# B&R Automation Studio project NAELD004C00R10L518F00 (part 41)

#### InputRef.var - Do Not Change!!!
```iecst
(*2021-08-01*)
(**)
(*General*)
VAR
	p_eAct : REFERENCE TO eHermesAction;
	p_udiRstErr : REFERENCE TO UDINT;
	p_bPrep : REFERENCE TO BOOL;
	p_bEn : REFERENCE TO BOOL;
	p_bDis : REFERENCE TO BOOL;
END_VAR
(**)
(*Configuration*)
VAR
	p_tyParam : REFERENCE TO tyHermesDSParam;
	p_sIPAddr : REFERENCE TO STRING[15];
	pa_usiMacAddr : REFERENCE TO ARRAY[0..5] OF USINT;
	p_tyDTStructure : REFERENCE TO DTStructure;
	p_dtCurrDT : REFERENCE TO DATE_AND_TIME;
	p_sMcId : REFERENCE TO STRING[80];
END_VAR
(**)
(*Input*)
VAR
	p_bRdySnd : REFERENCE TO BOOL;
	p_bSndCompl : REFERENCE TO BOOL;
	p_bSndIncompl : REFERENCE TO BOOL;
	p_bSndNotStart : REFERENCE TO BOOL;
	p_bBAWidthEn : REFERENCE TO BOOL; (*Board Available Check Width*)
	p_bBASltEn : REFERENCE TO BOOL; (*Board Available Check Slot*)
	p_bBFWidthEn : REFERENCE TO BOOL; (*Board Forecast Check Width*)
	p_bBFSltEn : REFERENCE TO BOOL; (*Board Forecast Check Slot*)
	p_sRecipeNm : REFERENCE TO STRING[254];
	p_sForecastId : REFERENCE TO STRING[80];
	p_sBoardId : REFERENCE TO STRING[36];
	p_sInterfaceId : REFERENCE TO STRING[80];
	p_sVersion : REFERENCE TO STRING[7];
	p_eFailedBoard : REFERENCE TO eHermesFailedBoard;
	p_eFlippedBoard : REFERENCE TO eHermesFlippedBoard;
	p_sTopBarcode : REFERENCE TO STRING[254];
	p_sBottomBarcode : REFERENCE TO STRING[254];
	p_rLength : REFERENCE TO REAL;
	p_rThickness : REFERENCE TO REAL;
	p_rConveyorSpeed : REFERENCE TO REAL;
	p_rTopClearanceHeight : REFERENCE TO REAL;
	p_rBottomClearanceHeight : REFERENCE TO REAL;
	p_rWeight : REFERENCE TO REAL;
	p_sWorkOrderId : REFERENCE TO STRING[80];
	p_sBatchId : REFERENCE TO STRING[80];
	p_diWidthInUM : REFERENCE TO DINT;
	p_diMinSltValue : REFERENCE TO DINT;
	p_diMaxSltValue : REFERENCE TO DINT;
	p_diPitch : REFERENCE TO DINT;
	p_diTtlSlt : REFERENCE TO DINT;
	p_diSltToSltInUM : REFERENCE TO DINT;
	p_udiSndBffrSize : REFERENCE TO UDINT;
	p_udiRcvBffrSize : REFERENCE TO UDINT;
	p_udiAliveIdleTimeInSec : REFERENCE TO UDINT;
	p_tConnTimeOut : REFERENCE TO TIME;
	p_diTransferInTO : REFERENCE TO DINT;
	pa_tyXMLTableDataBrdAvl : REFERENCE TO ARRAY[0..200] OF tyXMLTableDat;
	p_iXMLTableDataBrdAvlTtlIdx : REFERENCE TO INT;
	p_bNewBrdAvlFirstZone : REFERENCE TO BOOL;
	p_bNewBrdAvlLastZone : REFERENCE TO BOOL;
	p_bOpsRun : REFERENCE TO BOOL;
	p_bInterruptSen : REFERENCE TO BOOL;
	p_udiFileKeepDay : REFERENCE TO UDINT;
	p_udiRetainDataAddr : REFERENCE TO UDINT;
	p_udiRetainDataLen : REFERENCE TO UDINT;
	p_sRetainFileName : REFERENCE TO STRING[80];
	p_sProgNm : REFERENCE TO STRING[15];
	p_bNtSettingsLoadDone : REFERENCE TO BOOL;
	p_bRmtPrep : REFERENCE TO BOOL;
	p_bRmtEn : REFERENCE TO BOOL;
	p_bSvyPrep : REFERENCE TO BOOL;
	p_bSvyEn : REFERENCE TO BOOL;
	p_bOpsGConv1HvBrd : REFERENCE TO BOOL;
	p_bAllZonesEmpty : REFERENCE TO BOOL;
	p_bFirstZoneHaveBoard : REFERENCE TO BOOL;
	p_tyUSBoardArrivedData : REFERENCE TO tyHermesBoardAvailable;
	p_rMcCycleTm : REFERENCE TO REAL;
	p_rAWCycleTm : REFERENCE TO REAL;
	p_bInitDone : REFERENCE TO BOOL;
	p_tyHermesConfiguration : REFERENCE TO tyHermesConfiguration;
	p_bUSHermesStopTransport : REFERENCE TO BOOL;
	p_bRcvBoardInfo : REFERENCE TO BOOL;
	p_tyBoardInfoData : REFERENCE TO tyHermesSendBoardInfo;
	p_tySendWorkOrderData : REFERENCE TO tyHermesSendWorkOrderInfo;
	p_bUSHermesTransporting : REFERENCE TO BOOL;
	p_bReplyWorkOrderInfo : REFERENCE TO BOOL;
	p_bSendBoardForecast : REFERENCE TO BOOL;
	p_bClearWorkOrder : REFERENCE TO BOOL;
	p_bFirstZoneEndSen : REFERENCE TO BOOL;
	p_bNewProduct : REFERENCE TO BOOL;
	p_bNewWidth : REFERENCE TO BOOL;
	p_bInternalUse : REFERENCE TO BOOL;
	p_sInternalRcv : REFERENCE TO STRING[65535];
	p_tyDI : REFERENCE TO tyDigitalInput;
	p_usiProdRcpCurrRcp1McMod : REFERENCE TO USINT;
	p_usiSelProdRcpStep : REFERENCE TO USINT;
END_VAR
(**)
(*Dummy*)
VAR
	p_sFoundAddressTop : REFERENCE TO STRING[254];
	p_sFoundAddressBottom : REFERENCE TO STRING[254];
END_VAR
```

#### Local.var - Do Not Change!!!
```iecst
(*2021-08-01*)
(**)
(*Local Action, State & Status*)
VAR
	eAct : eHermesAction := HermesActIdle;
	eStat : eHermesAction := HermesActIdle;
	eMainStatus : eFBStatus := Idle;
	eStatus : eFBStatus := Idle;
	eStatus1 : eFBStatus := Idle;
	eStatus2 : eFBStatus := Idle;
	eStatus3 : eFBStatus := Idle;
	udiStatus : UDINT := 0;
	udiStatus1 : UDINT := 0;
	udiStatus2 : UDINT := 0;
	udiStatus3 : UDINT := 0;
	udiStatus4 : UDINT := 0;
	sStatTxt : STRING[200] := '';
	a_sStatText : ARRAY[0..50] OF STRING[200] := ['Idling','Background Starting Operations','Background Stopping Operations','Deleting Old Log File','Creating Directory','Writing Retain File','Reading Retain File','Saving Configuration',43('')];
END_VAR
(**)
(*Local Alarm*)
VAR
	tyAlmData : tyAlmDat;
	tyAlmData1 : tyAlmDat;
	tyAlmData2 : tyAlmDat;
	tyAlmData3 : tyAlmDat;
	tyAlmData4 : tyAlmDat;
	a_tyAlmText : ARRAY[10000..10199] OF tyAlmTxt := [(sAlmText:='Invalid Ident While Creating Server',sRcyText:='Problem Occurred In The TCP/IP Connection. Check The Connection And Try To Reconnect.'),(sAlmText:='Setting Keep Alive Interval Time Error While Creating Server',sRcyText:='Unable To Establish Connection Between Machine. Check For Setting And Resume Operation.'),(sAlmText:='Setting Keep Alive Idle Time Error While Creating Server',sRcyText:='Unable To Establish Connection Between Machine. Check For Setting And Resume Operation.'),(sAlmText:='Setting Keep Alive Count Error While Creating Server',sRcyText:='Unable To Establish Connection Between Machine. Check For Setting And Resume Operation.'),(sAlmText:='Setting Keep Alive Error While Creating Server',sRcyText:='Unable To Establish Connection Between Machine. Check For Setting And Resume Operation.'),(sAlmText:='Setting Receive Buffer Error While Creating Server',sRcyText:='Unable To Establish Connection Between Machine. Check For Setting And Resume Operation.'),(sAlmText:='Setting Send Buffer Error While Creating Server',sRcyText:='Unable To Establish Connection Between Machine. Check For Setting And Resume Operation.'),(sAlmText:='Setting No Waiting Error While Creating Server',sRcyText:='Unable To Establish Connection Between Machine. Check For Setting And Resume Operation.'),(sAlmText:='TCP Open Port Error While Creating Server',sRcyText:='Problem Occurred In The TCP/IP Connection. Check The Connection And Try To Reconnect.'),(sAlmText:='Closing TCP Error While Creating Server',sRcyText:='Problem Occurred In The TCP/IP Connection. Check The Connection And Try To Reconnect.'),(sAlmText:='Invalid Ident While Listening Client',sRcyText:='There Was A Problem Connecting To The Server. The Server May Not Exist or It is Unavailable At This Time. Check The Connection and Try Again.'),0,(sAlmText:='DS Hermes Connection Lost',sRcyText:='There Was A Problem Connecting To The Server. The Server May Not Exist or It is Unavailable At This Time. Check The Connection and Try Again.'),0,(sAlmText:='Invalid Ident While Receiving Data',sRcyText:='Problem Occurred In The TCP/IP Connection. Check The Connection And Try To Reconnect.'),(sAlmText:='TCP Receive Data Error While Receiving Data',sRcyText:='Problem Occurred In The TCP/IP Connection. Check The Connection And Try To Reconnect.'),(sAlmText:='Receive BoardAvailable While Downstream In Not Connected State',sRcyText:='Receive Illegal Message.'),(sAlmText:='Receive RevokeBoardAvailable While Downstream In Not Connected State',sRcyText:='Receive Illegal Message.'),(sAlmText:='Receive MachineReady While Downstream In Not Connected State',sRcyText:='Receive Illegal Message.'),(sAlmText:='Receive RevokeMachineReady While Downstream In Not Connected State',sRcyText:='Receive Illegal Message.'),(sAlmText:='Receive StartTransport While Downstream In Not Connected State',sRcyText:='Receive Illegal Message.'),(sAlmText:='Receive StopTransport While Downstream In Not Connected State',sRcyText:='Receive Illegal Message.'),(sAlmText:='Receive TransportFinished While Downstream In Not Connected State',sRcyText:='Receive Illegal Message.'),(sAlmText:='Receive BoardForecast While Downstream In Not Connected State',sRcyText:='Receive Illegal Message.'),(sAlmText:='Receive ServiceDescription While Downstream In Service Description State',sRcyText:='Receive Illegal Message.'),(sAlmText:='Receive BoardAvailable While Downstream In Service Description State',sRcyText:='Receive Illegal Message.'),(sAlmText:='Receive RevokeBoardAvailable While Downstream In Service Description State',sRcyText:='Receive Illegal Message.'),(sAlmText:='Receive MachineReady While Downstream In Service Description State',sRcyText:='Receive Illegal Message.'),(sAlmText:='Receive RevokeMachineReady While Downstream In Service Description State',sRcyText:='Receive Illegal Message.'),(sAlmText:='Receive StartTransport While Downstream In Service Description State',sRcyText:='Receive Illegal Message.'),(sAlmText:='Receive StopTransport While Downstream In Service Description State',sRcyText:='Receive Illegal Message.'),(sAlmText:='Receive TransportFinished While Downstream In Service Description State',sRcyText:='Receive Illegal Message.'),(sAlmText:='Receive BoardForecast While Downstream In Service Description State',sRcyText:='Receive Illegal Message.'),(sAlmText:='Receive ServiceDescription While Downstream In Not Available Not Ready State',sRcyText:='Receive Illegal Message.'),(sAlmText:='Receive BoardAvailable While Downstream In Not Available Not Ready State',sRcyText:='Receive Illegal Message.'),(sAlmText:='Receive RevokeBoardAvailable While Downstream In Not Available Not Ready State',sRcyText:='Receive Illegal Message.'),(sAlmText:='Receive RevokeMachineReady While Downstream In Not Available Not Ready State',sRcyText:='Receive Illegal Message.'),(sAlmText:='Receive StartTransport While Downstream In Not Available Not Ready State',sRcyText:='Receive Illegal Message.'),(sAlmText:='Receive StopTransport While Downstream In Not Available Not Ready State',sRcyText:='Receive Illegal Message.'),(sAlmText:='Receive TransportFinished While Downstream In Not Available Not Ready State',sRcyText:='Receive Illegal Message.'),(sAlmText:='Receive BoardForecast While Downstream In Not Available Not Ready State',sRcyText:='Receive Illegal Message.'),(sAlmText:='Receive ServiceDescription While Downstream In Board Available State',sRcyText:='Receive Illegal Message.'),(sAlmText:='Receive BoardAvailable While Downstream In Board Available State',sRcyText:='Receive Illegal Message.'),(sAlmText:='Receive RevokeBoardAvailable While Downstream In Board Available State',sRcyText:='Receive Illegal Message.'),(sAlmText:='Receive RevokeMachineReady While Downstream In Board Available State',sRcyText:='Receive Illegal Message.'),(sAlmText:='Receive StartTransport While Downstream In Board Available State',sRcyText:='Receive Illegal Message.'),(sAlmText:='Receive StopTransport While Downstream In Board Available State',sRcyText:='Receive Illegal Message.'),(sAlmText:='Receive TransportFinished While Downstream In Board Available State',sRcyText:='Receive Illegal Message.'),(sAlmText:='Receive BoardForecast While Downstream In Board Available State',sRcyText:='Receive Illegal Message.'),(sAlmText:='Receive ServiceDescription While Downstream In Machine Ready State',sRcyText:='Receive Illegal Message.'),(sAlmText:='Receive BoardAvailable While Downstream In Machine Ready State',sRcyText:='Receive Illegal Message.'),(sAlmText:='Receive RevokeBoardAvailable While Downstream In Machine Ready State',sRcyText:='Receive Illegal Message.'),(sAlmText:='Receive MachineReady While Downstream In Machine Ready State',sRcyText:='Receive Illegal Message.'),(sAlmText:='Receive StopTransport While Downstream In Machine Ready State',sRcyText:='Receive Illegal Message.'),(sAlmText:='Receive TransportFinished While Downstream In Machine Ready State',sRcyText:='Receive Illegal Message.'),(sAlmText:='Receive BoardForecast While Downstream In Machine Ready State',sRcyText:='Receive Illegal Message.'),(sAlmText:='Receive ServiceDescription While Downstream In Available And Ready State',sRcyText:='Receive Illegal Message.'),(sAlmText:='Receive BoardAvailable While Downstream In Available And Ready State',sRcyText:='Receive Illegal Message.'),(sAlmText:='Receive RevokeBoardAvailable While Downstream In Available And Ready State',sRcyText:='Receive Illegal Message.'),(sAlmText:='Receive MachineReady While Downstream In Available And Ready State',sRcyText:='Receive Illegal Message.'),(sAlmText:='Receive StopTransport While Downstream In Available And Ready State',sRcyText:='Receive Illegal Message.'),(sAlmText:='Receive TransportFinished While Downstream In Available And Ready State',sRcyText:='Receive Illegal Message.'),(sAlmText:='Receive BoardForecast While Downstream In Available And Ready State',sRcyText:='Receive Illegal Message.'),(sAlmText:='Receive ServiceDescription While Downstream In Transporting State',sRcyText:='Receive Illegal Message.'),(sAlmText:='Receive BoardAvailable While Downstream In Transporting State',sRcyText:='Receive Illegal Message.'),(sAlmText:='Receive RevokeBoardAvailable While Downstream In Transporting State',sRcyText:='Receive Illegal Message.'),(sAlmText:='Receive MachineReady While Downstream In Transporting State',sRcyText:='Receive Illegal Message.'),(sAlmText:='Receive RevokeMachineReady While Downstream In Transporting State',sRcyText:='Receive Illegal Message.'),(sAlmText:='Receive StartTransport While Downstream In Transporting State',sRcyText:='Receive Illegal Message.'),(sAlmText:='Receive TransportFinished While Downstream In Transporting State',sRcyText:='Receive Illegal Message.'),(sAlmText:='Receive BoardForecast While Downstream In Transporting State',sRcyText:='Receive Illegal Message.'),(sAlmText:='Receive ServiceDescription While In Transport Finished State',sRcyText:='Receive Illegal Message.'),(sAlmText:='Receive BoardAvailable While In Transport Finished State',sRcyText:='Receive Illegal Message.'),(sAlmText:='Receive RevokeBoardAvailable While In Transport Finished State',sRcyText:='Receive Illegal Message.'),(sAlmText:='Receive MachineReady While In Transport Finished State',sRcyText:='Receive Illegal Message.'),(sAlmText:='Receive RevokeMachineReady While In Transport Finished State',sRcyText:='Receive Illegal Message.'),(sAlmText:='Receive StartTransport While In Transport Finished State',sRcyText:='Receive Illegal Message.'),(sAlmText:='Receive TransportFinished While In Transport Finished State',sRcyText:='Receive Illegal Message.'),(sAlmText:='Receive BoardForecast While In Transport Finished State',sRcyText:='Receive Illegal Message.'),(sAlmText:='Receive ServiceDescription While Downstream In Transport Stopped State',sRcyText:='Receive Illegal Message.'),(sAlmText:='Receive BoardAvailable While Downstream In Transport Stopped State',sRcyText:='Receive Illegal Message.'),(sAlmText:='Receive RevokeBoardAvailable While Downstream In Transport Stopped State',sRcyText:='Receive Illegal Message.'),(sAlmText:='Receive MachineReady While Downstream In Transport Stopped State',sRcyText:='Receive Illegal Message.'),(sAlmText:='Receive RevokeMachineReady While Downstream In Transport Stopped State',sRcyText:='Receive Illegal Message.'),(sAlmText:='Receive StartTransport While Downstream In Transport Stopped State',sRcyText:='Receive Illegal Message.'),(sAlmText:='Receive StopTransport While Downstream In Transport Stopped State',sRcyText:='Receive Illegal Message.'),(sAlmText:='LaneId Mismatch While Checking Service Description',sRcyText:='The LaneId Value Does Not Match. Change The Value And Resend The Value.'),(sAlmText:='MachineId Missing While Checking Service Description',sRcyText:='Missing Input Value For MachineId. Fill Up The Value And Resend.'),(sAlmText:='LandId Out Of Range While Checking Service Description',sRcyText:='LaneId Does Not Fall Within The Expected Range.'),(sAlmText:='LandId Missing While Checking Service Description',sRcyText:='Missing Input Value For LaneId. Fill Up The Value And Resend.'),(sAlmText:='Version Missing While Checking Service Description',sRcyText:='Missing Input Value For Version. Fill Up The Value And Resend.'),(sAlmText:='SupportedFeatures Missing While Checking Service Description',sRcyText:='Missing Input Value For SupportedFeatures. Fill Up The Value And Resend.'),(sAlmText:='NotificationCode Out Of Range While Checking Notification',sRcyText:='NotificationCode Does Not Fall Within The Expected Range.'),(sAlmText:='NotificationCode Missing While Checking Notification',sRcyText:='Missing Input Value For NotificationCode. Fill Up The Value And Resend.'),(sAlmText:='Severity Missing While Checking Notification',sRcyText:='Missing Input Value For Severity. Fill Up The Value And Resend.'),(sAlmText:='Description Missing While Checking Notification',sRcyText:='Missing Input Value For Description. Fill Up The Value And Resend.'),2((0)),(sAlmText:='FailedBoard Missing While Checking Machine Ready',sRcyText:='Missing Input Value For FailedBoard. Fill Up The Value And Resend.'),(sAlmText:='TransferState Missing While Checking Stop Transport',sRcyText:='Missing Input Value For TransferState. Fill Up The Value And Resend.'),(sAlmText:='BoardId Missing While Checking Stop Transport',sRcyText:='Missing Input Value For BoardId. Fill Up The Value And Resend.'),(sAlmText:='BoardId Missing While Checking Start Transport',sRcyText:='Missing Input Value For BoardId. Fill Up The Value And Resend.'),(sAlmText:='Barcode Missing While Checking Query Board Info',sRcyText:='Missing Input Value For BoardId. Fill Up The Value And Resend.'),(0),(sAlmText:='BoardId Mismatch While Checking Start Transport & Stop Transport',sRcyText:='The BoardId Value Does Not Match. Change The Value And Resend The Value.'),(sAlmText:='BoardId Missing While Checking Start Transport & Stop Transport',sRcyText:='Missing Input Value For BoardId. Fill Up The Value And Resend.'),(sAlmText:='Service Description Interchange Time Out',sRcyText:='Timeout Expired Before Operation Completed. Reset And Resume Operation.'),(sAlmText:='Transport Time Out',sRcyText:='Timeout Expired Before Operation Completed. Reset And Resume Operation.'),(sAlmText:='Receive TransportFinished While Downstream In Transport Stopped State',sRcyText:='Receive Illegal Message.'),(sAlmText:='Receive BoardForecast While Downstream In Transport Stopped State',sRcyText:='Receive Illegal Message.'),(sAlmText:='Stop Transport Request To Send From Downstream Hermes',sRcyText:='Sending Illegal Message.'),(sAlmText:='Get Directory Info Error While Deleting Old Log',sRcyText:='An Error Was Encountered While Getting Directory Info. Please Contact Nutek For A Possible Solution.'),(sAlmText:='Directory Read Error While Deleting Old Log',sRcyText:='An Error Was Encountered While Reading Directory. Please Contact Nutek For A Possible Solution.'),(sAlmText:='File Delete Error While Deleting Old Log',sRcyText:='An Error Was Encountered While Trying To Delete File. Please Contact Nutek For A Possible Solution.'),(sAlmText:='File Open Error While Reading Retain File',sRcyText:='An Error Was Encountered While Trying To Open File. Please Contact Nutek For A Possible Solution.'),(sAlmText:='File Read Error While Reading Retain File',sRcyText:='An Error Was Encountered While Trying To Read File. Please Contact Nutek For A Possible Solution.'),(sAlmText:='File Close Error While Reading Retain File',sRcyText:='An Error Was Encountered While Trying To Close File. Please Contact Nutek For A Possible Solution.'),(sAlmText:='File Open Error While Writing Retain File',sRcyText:='An Error Was Encountered While Trying To Open File. Please Contact Nutek For A Possible Solution.'),(sAlmText:='File Create Error While Writing Retain File',sRcyText:='An Error Was Encountered While Trying To Create File. Please Contact Nutek For A Possible Solution.'),(sAlmText:='File Write Error While Writing Retain File',sRcyText:='An Error Was Encountered While Trying To Write File. Please Contact Nutek For A Possible Solution.'),(sAlmText:='File Close Error While Writing Retain File',sRcyText:='An Error Was Encountered While Trying To Close File. Please Contact Nutek For A Possible Solution.'),(sAlmText:='Directory Does Not Exist While Writing Retain File',sRcyText:='The Directory Does Not Exist. Please Contact Nutek For A Possible Solution.'),10((0)),(sAlmText:='Check Alive Time Out',sRcyText:='Timeout Expired Before Operation Completed. Reset And Resume Operation.'),(sAlmText:='Waiting Check Alive Time Out',sRcyText:='Timeout Expired Before Operation Completed. Reset And Resume Operation.'),(sAlmText:='Check Alive Id Mismatch',sRcyText:='The Check Alive Id Value Does Not Match. Change The Value And Resend The Value.'),(sAlmText:='Machine Ready Request To Send From Downstream Hermes',sRcyText:='Sending Illegal Message.'),(sAlmText:='Revoke Machine Ready Request To Send From Downstream Hermes',sRcyText:='Sending Illegal Message.'),(sAlmText:='Start Transport Request To Send From Downstream Hermes',sRcyText:='Sending Illegal Message.'),(sAlmText:='Set Configuration Request To Send From Downstream Hermes',sRcyText:='Sending Illegal Message.'),(sAlmText:='Get Configuration Request To Send From Downstream Hermes',sRcyText:='Sending Illegal Message.'),(sAlmText:='Current Configuration Request To Send From Downstream Hermes',sRcyText:='Sending Illegal Message.'),(sAlmText:='Board Forecast Request To Send From Downstream Hermes',sRcyText:='Sending Illegal Message.'),(sAlmText:='Query Board Info Request To Send From Downstream Hermes',sRcyText:='Sending Illegal Message.'),(sAlmText:='Invalid Ident While Sending Data',sRcyText:='Invalid Ident Value.'),(sAlmText:='TCP Retry Send Data Error While Sending Data',sRcyText:='Problem Occurred In The TCP/IP Connection. Check The Connection And Try To Reconnect.'),(sAlmText:='TCP Send Data Error',sRcyText:='Problem Occurred In The TCP/IP Connection. Check The Connection And Try To Reconnect.'),(sAlmText:='Invalid Ident While Closing TCP',sRcyText:='Invalid Ident Value.'),(sAlmText:='Closing TCP Error',sRcyText:='Problem Occurred In The TCP/IP Connection. Check The Connection And Try To Reconnect.'),(sAlmText:='File Open Error While Writing Log',sRcyText:='An Error Was Encountered While Trying To Open File. Please Contact Nutek For A Possible Solution.'),(sAlmText:='File Create Error While Writing Log',sRcyText:='An Error Was Encountered While Trying To Create File. Please Contact Nutek For A Possible Solution.'),(sAlmText:='Get File Info Error While Writing Log',sRcyText:='An Error Was Encountered While Getting File Info. Please Contact Nutek For A Possible Solution.'),(sAlmText:='File Write Error While Writing Log',sRcyText:='An Error Was Encountered While Trying To Write File. Please Contact Nutek For A Possible Solution.'),(sAlmText:='File Close Error While Writing Log',sRcyText:='An Error Was Encountered While Trying To Close File. Please Contact Nutek For A Possible Solution.'),(sAlmText:='Directory Does Not Exist While Writing Log',sRcyText:='The Directory Does Not Exist.Please Contact Nutek For A Possible Solution.'),(sAlmText:='Invalid Ident While Closing TCP',sRcyText:='Invalid Ident Value.'),(sAlmText:='Closing TCP Error',sRcyText:='Problem Occurred In The TCP/IP Connection. Check The Connection And Try To Reconnect.'),0,(sAlmText:='Board Jam At Sensor After Transfer Interrupted',sRcyText:='Pull Back Board From Downstream Machine'),0,(sAlmText:='Send Board Info Request To Send From Downstream Hermes',sRcyText:='Sending Illegal Message.'),(sAlmText:='Query Work Order Info Request To Send From Downstream Hermes',sRcyText:='Sending Illegal Message.'),(sAlmText:='Send Work Order Info Request To Send From Downstream Hermes',sRcyText:='Sending Illegal Message.'),(sAlmText:='Board Arrived Request To Send From Downstream Hermes',sRcyText:='Sending Illegal Message.'),(sAlmText:='Board departed Request To Send From Downstream Hermes',sRcyText:='Sending Illegal Message.'),(sAlmText:='Forecast Id Mismatch While Checking BoardForecast & Machine Ready',sRcyText:='The ForecastId Value Does Not Match. Change The Value And Resend The Value.'),(sAlmText:='Product Type Id Mismatch While Checking BoardForecast & Machine Ready',sRcyText:='The ProductTypetId Value Does Not Match. Change The Value And Resend The Value.'),(sAlmText:='Width Mismatch While Checking BoardForecast & Machine Ready',sRcyText:='The Width Value Does Not Match. Change The Value And Resend The Value.'),(sAlmText:='Query Top Barcode and Bottom Barcode found from different Recipes',sRcyText:='Please Check or Scan Again the PCB Barcode'),32(0)];
END_VAR
(**)
(*Local Output*)
VAR
	bConnected : BOOL;
	bHandshakeDone : BOOL;
	bSendOk : BOOL;
	bSearchTop : BOOL;
	bSearchBottom : BOOL;
	bFoundIndex : BOOL;
	bFoundTop : BOOL;
	bFoundBottom : BOOL;
	bFoundNothing : BOOL;
	bNewChangeOver : BOOL;
	bSendBFId : BOOL;
	bRstSendBFId : BOOL;
	bUSRdy : BOOL;
	bDSRdy : BOOL;
	bUSGdRdy : BOOL;
	bDSGdRdy : BOOL;
	bTransporting : BOOL;
	bStopTransport : BOOL;
	sInternalSnd : STRING[65535];
	bTransportFinishedSnd : BOOL;
	tyBoardDepartedInfo : tyHermesBoardAvailable;
END_VAR
(**)
(*Local Input*)
VAR
	udiRstErr : UDINT := 0;
	bPrep : BOOL := TRUE;
	bEn : BOOL := TRUE;
	bDis : BOOL := FALSE;
	tyParam : tyHermesDSParam;
	sIPAddr : STRING[15] := '192.168.0.100';
	a_usiMacAddr : ARRAY[0..5] OF USINT := [6(0)];
	tyDTStructure : DTStructure := (year:=2020,month:=11,day:=11,wday:=05,hour:=21,minute:=28,second:=30,millisec:=123,microsec:=456);
	dtCurrDT : DATE_AND_TIME := DT#2019-02-23-12:30:50;
	bRdySnd : BOOL := FALSE;
	bSndCompl : BOOL := FALSE;
	bSndInCompl : BOOL := FALSE;
	bSndNotStart : BOOL := FALSE;
	bFirstZoneEndSen : BOOL;
	bBAWidthEn : BOOL := TRUE; (*Board Available Check Width*)
	bBASltEn : BOOL := TRUE; (*Board Available Check Slot*)
	bBFWidthEn : BOOL := TRUE; (*Board Forecast Check Width*)
	bBFSltEn : BOOL := FALSE; (*Board Forecst Check Slot*)
	sForecastId : {REDUND_UNREPLICABLE} STRING[80] := '';
	sBoardId : STRING[36] := '';
	sMcId : STRING[80] := '';
	sInterfaceId : STRING[80] := '';
	sVersion : STRING[7] := '1.3';
	eFailedBoard : eHermesFailedBoard := HermesUnknownBoard;
	sRecipeNm : STRING[254] := '';
	eFlippedBoard : eHermesFlippedBoard := HermesFlippedBoardUnknownSide;
	sTopBarcode : STRING[254] := '';
	sBottomBarcode : STRING[254] := '';
	rLength : REAL := 0;
	rThickness : REAL := 0;
	rConveyorSpeed : REAL := 0;
	rTopClearanceHeight : REAL := 0;
	rBottomClearanceHeight : REAL := 0;
	rWeight : REAL := 0;
	sWorkOrderId : STRING[80] := '';
	sBatchId : STRING[80] := '';
	diWidthInUM : DINT := 0;
	diMinSltValue : DINT := 0;
	diMaxSltValue : DINT := 0;
	diPitch : DINT := 0;
	diTtlSlt : DINT := 0;
	diSltToSltInUM : DINT := 0;
	udiSndBffrSize : UDINT := 65536;
	udiRcvBffrSize : UDINT := 65536;
	udiAliveIdleTimeInSec : UDINT := 5;
	tConnTimeOut : TIME := T#30s;
	diTransferInTO : DINT := 30000;
	a_tyXMLTableDataBrdAvl : ARRAY[0..200] OF tyXMLTableDat;
	iXMLTableDataBrdAvlTtlIdx : INT := 0;
	bNewBrdAvl1 : BOOL := FALSE;
	bNewBrdAvl2 : BOOL := FALSE;
	bOpsRun : BOOL := FALSE;
	bInterruptSen : BOOL := FALSE;
	udiFileKeepDay : UDINT := 30;
	sRetainFileName : STRING[80] := 'BoardData.dat';
	sProgNm : STRING[15] := 'DSHermes';
	bNtSettingsLoadDone : BOOL := TRUE;
	bRmtPrep : BOOL := FALSE;
	bRmtEn : BOOL := FALSE;
	bSvyPrep : BOOL := FALSE;
	bSvyEn : BOOL := FALSE;
	bAllZonesEmpty : BOOL := FALSE;
	bFirstZoneHaveBoard : BOOL := FALSE;
	bInternalUse : BOOL;
	sInternalRcv : STRING[65535];
	rMachineCycleTime : REAL := 6000;
	rAutoWidthCycleTime : REAL := 30000;
	tyHermesCurrConfiguration : tyHermesConfiguration;
	tyBoardInfoData : tyHermesSendBoardInfo;
	tyUSBoardArrivedData : tyHermesBoardAvailable;
	bUSHermesStopTransport : BOOL;
	bRcvBoardInfo : BOOL;
	bUSHermesTransporting : BOOL;
	bOpsGConv1HvBrd : BOOL;
END_VAR
(**)
(*Local*)
VAR
	bRstErr : BOOL;
	udiRstErrOld : UDINT;
	bInitDone : BOOL;
	bInitialDone : BOOL;
	bRun : BOOL;
	bStop : BOOL;
	bRstConnection : BOOL;
	bRstState : BOOL;
	udiSvrIdent : UDINT;
	udiClntIdent : UDINT;
	udiClntIdentExtra : UDINT;
	udiXMLTableWriteIdx : UDINT;
	udiMsgSendBffr : UDINT;
	udiSndMsgLen : UDINT;
	sSnd : STRING[65535];
	sRcv : STRING[65535];
	a_tyXMLTableDataRcv : ARRAY[0..200] OF tyXMLTableDat;
	a_tyXMLTableDataSnd : ARRAY[0..200] OF tyXMLTableDat;
	a_eMsgSend : ARRAY[0..50] OF eHermesMsgType;
	tyMsgTypeRcv : tyHermesMsgType;
	tyCheckAliveSnd : tyHermesCheckAlive;
	tyCheckAlivePingSnd : tyHermesCheckAlive;
	tyCheckAlivePongSnd : tyHermesCheckAlive;
	tyCheckAliveRcv : tyHermesCheckAlive;
	tyCheckAlivePingRcv : tyHermesCheckAlive;
	tyCheckAlivePongRcv : tyHermesCheckAlive;
	tyServiceDescriptionSnd : tyHermesServiceDescription;
	tyServiceDescriptionRcv : tyHermesServiceDescription;
	tyNotificationSnd : tyHermesNotification;
	tyNotificationRcv : tyHermesNotification;
	tyBoardAvailableRcv : tyHermesBoardAvailable;
	tyBoardAvailableSnd : tyHermesBoardAvailable;
	a_tyBoardDepartedInfo : ARRAY[0..49] OF tyHermesBoardAvailable;
	tyMachineReady : tyHermesMachineReady;
	tyStartTransport : tyHermesStartTransport;
	tyStopTransport : tyHermesStopTransport;
	tyTransportFinished : tyHermesTransportFinished;
	tySetConfiguration : tyHermesSetConfiguration;
	tyCurrentConfiguration : tyHermesCurrentConfiguration;
	tyBoardForecastRcv : tyHermesBoardForecast;
	tyBoardForecastSnd : tyHermesBoardForecast;
	tyQueryBoardInfo : tyHermesQueryBoardInfo;
	tySendBoardInfo : tyHermesSendBoardInfo;
	fbCreateSvr : fbTCPCreateSvr;
	fbListen : fbTCPListen;
	fbRcv : fbTCPRcv;
	fbSend : fbTCPSnd;
	fbCloseSvr : fbTCPClose;
	fbCloseClnt : fbTCPClose;
	fbParseXMLTable : fbHermesParseXMLTable;
	fbParseBrdAvlExternal : fbHermesParseXMLTable;
	fbCheckAlive : fbHermesCheckAlive;
	fbCheckAliveSendPing : fbHermesCheckAliveSendPing;
	fbCheckAliveRcvPing : fbHermesCheckAliveRcvPing;
	fbSequenceDS : fbHermesSequenceDS;
	fbSequenceTO : fbHermesSequenceTO;
	eStatOld : eHermesAction := HermesActIdle;
	tyParamOld : tyHermesDSParam;
	bFeatureBoardForecast : BOOL;
	bNewProduct : USINT;
	bNewWidth : BOOL;
	bSiemensNewProduct : BOOL;
	bTest888 : BOOL;
	idxBoardForecastId : INT := 0;
	idxBoardForecastNoId : INT := 0;
END_VAR
VAR RETAIN
	udiBAIndex : UDINT := 0;
END_VAR
VAR
	i : UDINT := 0;
	j : UDINT := 0;
	jj : UDINT := 0;
	udiTopTargetAddress : UDINT := 0;
	udiBottomTargetAddress : UDINT := 0;
	udiSizeOfAddress : UDINT := 0;
	udiTargetAddress : UDINT := 0;
	udiSizeAddress : UDINT := 0;
	udiFoundAddressTop : UDINT := 0;
	udiFoundRecipeTop : UDINT := 0;
	udiFoundRecipeFinal : UDINT := 0;
	udiFoundAddressBottom : UDINT := 0;
	udiFoundRecipeBottom : UDINT := 0;
	sSearchTop : STRING[254] := '';
	sSearchBottom : STRING[254] := '';
	udiLogCntr : UDINT := 1;
	udiWriteLogCntr : UDINT := 1;
	a_sLogList : ARRAY[1..10] OF STRING[65535];
	sDT : STRING[80];
	dtCurrDTTemp : DATE_AND_TIME;
	fbFileAppend1 : fbFileFullAppend;
	fbFileOldDel1 : fbFileOldDel;
	fbFileRead1 : fbFileFullRead;
	fbFileWrite1 : fbFileFullWrite;
	fbSendTm : TON;
	bFileNotFound : BOOL;
	udiRetainDataAddr : UDINT;
	udiRetainDataLen : UDINT;
	iWriteLogStep : INT := 0;
	fbDeleteLogTmr : TON := (PT:=T#24h);
	fbDlyTmr : TON := (PT:=T#5s);
	udiModuleNum : UDINT := 3351;
END_VAR
```

### RmtHermes.var - Change By Project
```iecst
(*2021-08-01*)
(**)
(*Action & State & Status*)
VAR
	p_RmtHermesStat : UDINT;
	p_RmtHermesStatus : UDINT;
	p_RmtHermesStatTxt : UDINT;
	p_RmtHermesAct : UDINT;
	p_RmtHermesMcParamAct : UDINT;
END_VAR
(**)
(*Alarm*)
VAR
	p_RmtHermesAlmData : UDINT;
	p_RmtHermesAlmData1 : UDINT;
	p_RmtHermesAlmData2 : UDINT;
	p_RmtHermesAlmData3 : UDINT;
	p_RmtHermesInfoData : UDINT;
END_VAR
(**)
(*Output*)
VAR
	p_RmtHermesFileNotFound : UDINT;
	p_RmtHermesConnected : UDINT;
	p_RmtHermesWriteConfig : UDINT;
	p_RmtHermesUpdateUIData : UDINT;
	p_RmtHermesSetConfiguration : UDINT;
	p_RmtHermesFoundIndexUS1 : UDINT;
	p_RmtHermesFoundIndexUS2 : UDINT;
	p_RmtHermesFoundIndexUS3 : UDINT;
	p_RmtHermesFoundIndexUS4 : UDINT;
	p_RmtHermesFoundIndexDS1 : UDINT;
	p_RmtHermesFoundIndexDS2 : UDINT;
	p_RmtHermesFoundIndexDS3 : UDINT;
	p_RmtHermesFoundIndexDS4 : UDINT;
	p_RmtHermesIndexUS1 : UDINT;
	p_RmtHermesIndexUS2 : UDINT;
	p_RmtHermesIndexUS3 : UDINT;
	p_RmtHermesIndexUS4 : UDINT;
	p_RmtHermesIndexDS1 : UDINT;
	p_RmtHermesIndexDS2 : UDINT;
	p_RmtHermesIndexDS3 : UDINT;
	p_RmtHermesIndexDS4 : UDINT;
END_VAR
```

### Program Logical/Hermes/RmtHermes (IEC, version 1.00.0) - 1.00.0 - NtHermes v5.00.0 , NtTCP v5.00.0 , NtMessage v5.00.0

#### Act_Alarm.st - Do Not Change!!!
```iecst
(** 2021-08-01 **)
ACTION Act_Alarm: //General

	//Error
	IF EDGEPOS(eStatus = Error) THEN

		tyAlmData.sProgNm		:= p_sProgNm;
		tyAlmData.udiCode		:= udiStatus;
		tyAlmData.eSeverity		:= AlmSeverityError;
		tyAlmData.udiRunTime	:= tyAlmData.udiRunTime + 1;
		tyAlmData.bAlm			:= TRUE;
		tyAlmData.udiModuleNum  := udiModuleNum;
		g_sRmtHermesProgNm		:= p_sProgNm;
		//Get Error Message
		IF tyAlmData.udiCode < 10000 OR tyAlmData.udiCode > 10199 THEN
			tyAlmData.sAlmMsg	:= 'Unknown';
			tyAlmData.sRcyMsg	:= 'Unknown';
		ELSE
			tyAlmData.sAlmMsg	:= a_tyAlmText[tyAlmData.udiCode].sAlmText;
			tyAlmData.sRcyMsg	:= a_tyAlmText[tyAlmData.udiCode].sRcyText;
		END_IF

		sStatTxt	:= tyAlmData.sAlmMsg;

	ELSIF bRstErr AND (tyAlmData.udiCode <> 0) THEN

		tyAlmData.udiCode	:= 0;
		tyAlmData.eSeverity	:= AlmSeverityNA;
		tyAlmData.sAlmMsg	:= '';
		tyAlmData.sRcyMsg	:= '';
		tyAlmData.bAlm			:= FALSE;
		sStatTxt	:= a_sStatText[eStat];

	END_IF

END_ACTION
```

#### Act_Alarm1.st - Do Not Change!!!
```iecst
(** 2021-08-01 **)
ACTION Act_Alarm1:

	//Error
	IF EDGEPOS(eStatus1 = Error) THEN

		tyAlmData1.sProgNm		:= p_sProgNm;
		tyAlmData1.udiCode		:= udiStatus1;
		tyAlmData1.eSeverity	:= AlmSeverityError;
		tyAlmData1.udiRunTime	:= tyAlmData1.udiRunTime + 1;
		tyAlmData1.bAlm			:= TRUE;
		tyAlmData1.udiModuleNum  := udiModuleNum;
		g_sRmtHermesProgNm		:= p_sProgNm;
		//Get Error Message
		IF tyAlmData1.udiCode < 10000 OR tyAlmData1.udiCode > 10199 THEN
			tyAlmData1.sAlmMsg	:= 'Unknown';
			tyAlmData1.sRcyMsg	:= 'Unknown';
		ELSE
			tyAlmData1.sAlmMsg	:= a_tyAlmText[tyAlmData1.udiCode].sAlmText;
			tyAlmData1.sRcyMsg	:= a_tyAlmText[tyAlmData1.udiCode].sRcyText;
		END_IF

		sStatTxt	:= tyAlmData1.sAlmMsg;

	ELSIF bRstErr AND (tyAlmData1.udiCode <> 0) THEN

		tyAlmData1.udiCode		:= 0;
		tyAlmData1.eSeverity	:= AlmSeverityNA;
		tyAlmData1.sAlmMsg		:= '';
		tyAlmData1.sRcyMsg		:= '';
		tyAlmData1.bAlm			:= FALSE;
		sStatTxt	:= a_sStatText[eStat];

	END_IF

END_ACTION
```

#### Act_Alarm2.st - Do Not Change!!!
```iecst
(** 2021-08-01 **)
ACTION Act_Alarm2:

	//Error
	IF EDGEPOS(eStatus2 = Error) THEN

		tyAlmData2.sProgNm		:= p_sProgNm;
		tyAlmData2.udiCode		:= udiStatus2;
		tyAlmData2.eSeverity	:= AlmSeverityError;
		tyAlmData2.udiRunTime	:= tyAlmData2.udiRunTime + 1;
		tyAlmData2.bAlm			:= TRUE;
		tyAlmData2.udiModuleNum  := udiModuleNum;
		g_sRmtHermesProgNm		:= p_sProgNm;
		//Get Error Message
		IF tyAlmData2.udiCode < 10000 OR tyAlmData2.udiCode > 10199 THEN
			tyAlmData2.sAlmMsg	:= 'Unknown';
			tyAlmData2.sRcyMsg	:= 'Unknown';
		ELSE
			tyAlmData2.sAlmMsg	:= a_tyAlmText[tyAlmData2.udiCode].sAlmText;
			tyAlmData2.sRcyMsg	:= a_tyAlmText[tyAlmData2.udiCode].sRcyText;
		END_IF

		sStatTxt	:= tyAlmData2.sAlmMsg;

	ELSIF bRstErr AND (tyAlmData2.udiCode <> 0) THEN

		tyAlmData2.udiCode		:= 0;
		tyAlmData2.eSeverity	:= AlmSeverityNA;
		tyAlmData2.sAlmMsg		:= '';
		tyAlmData2.sRcyMsg		:= '';
		tyAlmData2.bAlm			:= FALSE;
		sStatTxt	:= a_sStatText[eStat];

	END_IF

END_ACTION
```

#### Act_Alarm3.st - Do Not Change!!!
```iecst
(** 2021-08-01 **)
ACTION Act_Alarm3: //fbFileAppend1 Error

	//Error
	IF EDGEPOS(eStatus3 = Error) THEN

		tyAlmData3.sProgNm		:= p_sProgNm;
		tyAlmData3.udiCode		:= udiStatus3;
		tyAlmData3.eSeverity	:= AlmSeverityError;
		tyAlmData3.udiRunTime	:= tyAlmData3.udiRunTime + 1;
		tyAlmData3.bAlm			:= TRUE;
		tyAlmData3.udiModuleNum  := udiModuleNum;
		g_sRmtHermesProgNm		:= p_sProgNm;
		//Get Error Message
		IF tyAlmData3.udiCode < 10000 OR tyAlmData3.udiCode > 10199 THEN
			tyAlmData3.sAlmMsg	:= 'Unknown';
			tyAlmData3.sRcyMsg	:= 'Unknown';
		ELSE
			tyAlmData3.sAlmMsg	:= a_tyAlmText[tyAlmData3.udiCode].sAlmText;
			tyAlmData3.sRcyMsg	:= a_tyAlmText[tyAlmData3.udiCode].sRcyText;
		END_IF

		sStatTxt	:= tyAlmData3.sAlmMsg;

	ELSIF bRstErr AND (tyAlmData3.udiCode <> 0) THEN

		tyAlmData3.udiCode		:= 0;
		tyAlmData3.eSeverity	:= AlmSeverityNA;
		tyAlmData3.sAlmMsg		:= '';
		tyAlmData3.sRcyMsg		:= '';
		tyAlmData3.bAlm			:= FALSE;
		sStatTxt	:= a_sStatText[eStat];

	END_IF

END_ACTION
```

### SvyHermes.var - Change By Project
```iecst
(*2021-08-01*)
(**)
(*Action & State & Status*)
VAR
	p_SvyHermesStat : UDINT;
	p_SvyHermesStatus : UDINT;
	p_SvyHermesStatTxt : UDINT;
	p_SvyHermesAct : UDINT;
	p_SvyHermesMcParamAct : UDINT;
END_VAR
(**)
(*Alarm*)
VAR
	p_SvyHermesAlmData : UDINT;
	p_SvyHermesAlmData1 : UDINT;
	p_SvyHermesAlmData2 : UDINT;
	p_SvyHermesAlmData3 : UDINT;
	p_SvyHermesAlmData4 : UDINT;
	p_SvyHermesInfoData : UDINT;
	p_SvyHermesInfoData1 : UDINT;
	p_SvyHermesInfoData2 : UDINT;
	p_SvyHermesInfoData3 : UDINT;
	p_SvyHermesInfoData4 : UDINT;
END_VAR
(**)
(*Output*)
VAR
	p_SvyHermesConnected : UDINT;
	p_SvyHermesHandshakeDone : UDINT;
	p_SvyHermesFileNotFound : UDINT;
	p_SvyHermesSetConfiguration : UDINT;
	p_SvyHermesWriteConfig : UDINT;
	p_SvyHermesUpdateUIData : UDINT;
	p_SvyHermesInternalSnd : UDINT;
	p_SvyHermesWorkOrderId : UDINT;
	p_SvyHermesBatchId : UDINT;
	p_SvyHermesFoundIndexUS1 : UDINT;
	p_SvyHermesFoundIndexUS2 : UDINT;
	p_SvyHermesFoundIndexUS3 : UDINT;
	p_SvyHermesFoundIndexUS4 : UDINT;
	p_SvyHermesFoundIndexDS1 : UDINT;
	p_SvyHermesFoundIndexDS2 : UDINT;
	p_SvyHermesFoundIndexDS3 : UDINT;
	p_SvyHermesFoundIndexDS4 : UDINT;
	p_SvyHermesIndexUS1 : UDINT;
	p_SvyHermesIndexUS2 : UDINT;
	p_SvyHermesIndexUS3 : UDINT;
	p_SvyHermesIndexUS4 : UDINT;
	p_SvyHermesIndexDS1 : UDINT;
	p_SvyHermesIndexDS2 : UDINT;
	p_SvyHermesIndexDS3 : UDINT;
	p_SvyHermesIndexDS4 : UDINT;
	p_RcvBoardInfoOk : UDINT;
	p_ReplyWorkOrderInfo : UDINT;
	p_SendBoardForecast : UDINT;
	p_ClearWorkOrder : UDINT;
	p_NewIncomingBoard : UDINT;
	p_QueryBypassWorkOrder : UDINT;
	p_ReplyBypassWorkOrderInfo : UDINT;
	p_ReqLoaderWidthInUM : UDINT;
	p_RcvWorkOrderInfo1 : UDINT;
	p_SndWorkOrderInfo : UDINT;
	p_SvyHermesBypassSendWOData : UDINT;
	p_SvyHermesSendWorkOrderData : UDINT;
	p_SvyHermesSendWorkOrderDataRcv : UDINT;
END_VAR
(**)
VAR
	p_SvyHermesMagAccOrder : UDINT;
	p_SvyHermesMagGUID : UDINT;
	p_SvyHermesMagOrderPos : UDINT;
END_VAR
```

### Program Logical/Hermes/SvyHermes (IEC) - 1.00.1 - NtHermes v5.00.4 , NtTCP v5.00.2 , NtMessage v5.00.1

#### InputRef.var
```iecst
(*2021-08-01*)
(**)
(*Configuration*)
VAR
	p_tyParam : REFERENCE TO tyHermesSvyParam;
	p_sIPAddr : REFERENCE TO STRING[15];
	pa_usiMacAddr : REFERENCE TO ARRAY[0..5] OF USINT;
	p_tyDTStructure : REFERENCE TO DTStructure;
	p_dtCurrDT : REFERENCE TO DATE_AND_TIME;
	p_sMcId : REFERENCE TO STRING[80];
END_VAR
(**)
(*General*)
VAR
	p_eAct : REFERENCE TO eHermesAction;
	p_udiRstErr : REFERENCE TO UDINT;
	p_bPrep : REFERENCE TO BOOL;
	p_bEn : REFERENCE TO BOOL;
	p_bDis : REFERENCE TO BOOL;
END_VAR
(**)
(*Input*)
VAR
	p_sRecipeNm : REFERENCE TO STRING[254];
	p_sMagazineId : REFERENCE TO STRING[80];
	p_iSlotId : REFERENCE TO INT;
	p_eBoardTransfer1 : REFERENCE TO eHermesBoardTransfer;
	p_eBoardTransfer2 : REFERENCE TO eHermesBoardTransfer;
	p_eBoardTransfer3 : REFERENCE TO eHermesBoardTransfer;
	p_eBoardTransfer4 : REFERENCE TO eHermesBoardTransfer;
	p_sBarcode : REFERENCE TO STRING[254];
	p_sVersion : REFERENCE TO STRING[7];
	p_udiSndBffrSize : REFERENCE TO UDINT;
	p_udiRcvBffrSize : REFERENCE TO UDINT;
	p_udiAliveIdleTimeInSec : REFERENCE TO UDINT;
	p_tConnTimeOut : REFERENCE TO TIME;
	p_diTransferInTO : REFERENCE TO DINT;
	p_bNewBrdAvlLastZone : REFERENCE TO BOOL;
	p_bOpsRun : REFERENCE TO BOOL;
	p_udiFileKeepDay : REFERENCE TO UDINT;
	p_sConfigFileName : REFERENCE TO STRING[80];
	p_sProgNm : REFERENCE TO STRING[15];
	p_bNtSettingsLoadDone : REFERENCE TO BOOL;
	p_bSvyPrep : REFERENCE TO BOOL;
	p_bSvyEn : REFERENCE TO BOOL;
	p_bQueryWorkOrderInfo : REFERENCE TO BOOL;
	p_tyHermesConfiguration : REFERENCE TO tyHermesConfiguration;
	p_bUSHermesStopTransport1 : REFERENCE TO BOOL;
	p_bUSHermesStopTransport2 : REFERENCE TO BOOL;
	p_bUSHermesStopTransport3 : REFERENCE TO BOOL;
	p_bUSHermesStopTransport4 : REFERENCE TO BOOL;
	p_tyUSBoardArrived1 : REFERENCE TO tyHermesBoardAvailable;
	p_tyUSBoardArrived2 : REFERENCE TO tyHermesBoardAvailable;
	p_tyUSBoardArrived3 : REFERENCE TO tyHermesBoardAvailable;
	p_tyUSBoardArrived4 : REFERENCE TO tyHermesBoardAvailable;
	p_bDSHermesTransportFinished1 : REFERENCE TO BOOL;
	p_bDSHermesTransportFinished2 : REFERENCE TO BOOL;
	p_bDSHermesTransportFinished3 : REFERENCE TO BOOL;
	p_bDSHermesTransportFinished4 : REFERENCE TO BOOL;
	p_tyDSBoardDeparted1 : REFERENCE TO tyHermesBoardAvailable;
	p_tyDSBoardDeparted2 : REFERENCE TO tyHermesBoardAvailable;
	p_tyDSBoardDeparted3 : REFERENCE TO tyHermesBoardAvailable;
	p_tyDSBoardDeparted4 : REFERENCE TO tyHermesBoardAvailable;
	p_tyUSBoardAvailableRcv : REFERENCE TO tyHermesBoardAvailable;
	p_tyUSBoardForecastRcv : REFERENCE TO tyHermesBoardForecast;
	p_udiRetainDataAddr : REFERENCE TO UDINT;
	p_udiRetainDataLen : REFERENCE TO UDINT;
	p_udiLoaderRetainDataAddr0 : REFERENCE TO UDINT;
	p_udiLoaderRetainDataLen0 : REFERENCE TO UDINT;
	p_udiLoaderRetainDataAddr1 : REFERENCE TO UDINT;
	p_udiLoaderRetainDataLen1 : REFERENCE TO UDINT;
	p_udiBypassRetainDataAddr0 : REFERENCE TO UDINT;
	p_udiBypassRetainDataLen0 : REFERENCE TO UDINT;
	p_sInfoMsg : REFERENCE TO STRING[200];
	p_sInfoMsg1 : REFERENCE TO STRING[200];
	p_sInfoMsg2 : REFERENCE TO STRING[200];
	p_sInfoMsg3 : REFERENCE TO STRING[200];
	p_sInfoMsg4 : REFERENCE TO STRING[200];
	p_eMcParamStatus : REFERENCE TO eFBStatus;
	p_eMcParamStat : REFERENCE TO eMcParamAction;
	p_eHermesStatus : REFERENCE TO eFBStatus;
	p_eHermesStat : REFERENCE TO eHermesAction;
	p_bAllZonesEmpty : REFERENCE TO BOOL;
	p_bDeleteWorkOrder : REFERENCE TO BOOL;
	p_bFirstMcIntheLine : REFERENCE TO BOOL;
	p_sRetainFileName : REFERENCE TO STRING[80];
	p_sRetainFileName1 : REFERENCE TO STRING[80];
	p_sRetainFileName2 : REFERENCE TO STRING[80];
	p_sRetainFileName3 : REFERENCE TO STRING[80];
	p_sInternalRcv : REFERENCE TO STRING[65535];
	p_bInternalUse : REFERENCE TO BOOL;
	p_bAcceptCondition : REFERENCE TO BOOL;
	p_tyProdRcpCurrRcp : REFERENCE TO tyProdRcpParam;
	p_bLinkDIPresentSen : REFERENCE TO BOOL;
	p_tyDI : REFERENCE TO tyDigitalInput;
	p_bOpsConvWaitForTopUpBrd : REFERENCE TO BOOL;
	p_bOpsConvTopUpBrdReq : REFERENCE TO BOOL;
	p_bSendBFId : REFERENCE TO BOOL;
	p_bUSHermesUSRdy : REFERENCE TO BOOL;
	p_bUITopUpBrdRdy : REFERENCE TO BOOL;
	p_usiSelProdRcpStep : REFERENCE TO USINT;
	p_bLinkStepStackMode : REFERENCE TO BOOL;
	p_usiLinkProdRcpCurrRcpMcMod : REFERENCE TO USINT;
	p_eLinkMcParamUSCommMod : REFERENCE TO eMcSetCommMod;
END_VAR
```

#### InputRef_Link.var
```iecst
(*2021-08-01*)
(**)
VAR
	p_bLinkStartupRun : REFERENCE TO BOOL;
	p_bLinkOpsMagConvLD1QueryWO : REFERENCE TO BOOL;
	p_bLinkOpsMagConvLD2QueryWO : REFERENCE TO BOOL;
	p_bLinkOpsMagConvLD3QueryWO : REFERENCE TO BOOL;
	p_eLinkCustomerReq : REFERENCE TO eCustomer;
	p_bUIDeleteWorkOrder : REFERENCE TO BOOL;
	p_bAutoRcpCurrDeleteSendWO : REFERENCE TO BOOL;
	bHermesRun : BOOL;
	bHermesStop : BOOL;
END_VAR
(**)
VAR
	bLifterEmpty : BOOL;
	tySendWorkOrderInfoAccPublish : BOOL;
	bReplyWorkOrderInfo : BOOL;
	bReplyBypassWorkOrderInfo : BOOL;
	bRcvBoardInfoOk : BOOL;
	bRetainNewAcc : BOOL;
	bSendBoardForecast : BOOL;
	bClearWorkOrder : BOOL;
	pa_tyLinkXMLTableDataBrdAvl1 : REFERENCE TO ARRAY[0..200] OF tyXMLTableDat;
	p_iLinkXMLTableDataBrdAvlTtlIdx1 : REFERENCE TO INT;
	bNewIncomingBoard : BOOL;
	sUSBarcode : STRING[254];
	bQueryloaderWorkOrder : BOOL;
	bQueryBypassWorkOrder : BOOL;
	bRcvWorkBypassOrderInfo : BOOL;
	bManualQueryWO : BOOL;
	p_sHermesBrdId : REFERENCE TO STRING[36];
END_VAR
(*Loader Prop.*)
VAR
	p_diBuffer1Slt : REFERENCE TO DINT;
	p_diBuffer2Slt : REFERENCE TO DINT;
	p_diBuffer3Slt : REFERENCE TO DINT;
	p_bConvHvBrd : REFERENCE TO BOOL;
	p_bPullerRetRS : REFERENCE TO BOOL;
	p_eOpsTravLifLDPosGo : REFERENCE TO eTravLifLDPos;
	p_tyAutoRcpTravLif : REFERENCE TO tyBoardProperty;
END_VAR
```

#### Local.var
```iecst
(*2021-08-01*)
(**)
(*Local Action, State & Status*)
VAR
	eAct : eHermesAction := HermesActIdle;
	eStat : eHermesAction := HermesActIdle;
	eHermesAct : eHermesAction;
	eMcParamAct : eMcParamAction;
	eMainStatus : eFBStatus := Idle;
	eStatus : eFBStatus := Idle;
	eStatus1 : eFBStatus := Idle;
	eStatus2 : eFBStatus := Idle;
	eStatus3 : eFBStatus := Idle;
	udiStatus : UDINT := 0;
	udiStatus1 : UDINT := 0;
	udiStatus2 : UDINT := 0;
	udiStatus3 : UDINT := 0;
	udiStatus4 : UDINT := 0;
	udiStatus5 : UDINT;
	sStatTxt : STRING[200] := '';
	a_sStatText : ARRAY[0..50] OF STRING[200] := ['Idling','Background Starting Operations','Background Stopping Operations','Deleting Old Log File','Creating Directory','Writing Retain File','Reading Retain File','Saving Configuration',43('')];
END_VAR
(**)
(*Local Alarm*)
VAR
	tyAlmData : tyAlmDat;
	tyAlmData1 : tyAlmDat;
	tyAlmData2 : tyAlmDat;
	tyAlmData3 : tyAlmDat;
	tyAlmData4 : tyAlmDat;
	tyInfoData : tyAlmDat;
	tyInfoData1 : tyAlmDat;
	tyInfoData2 : tyAlmDat;
	tyInfoData3 : tyAlmDat;
	tyInfoData4 : tyAlmDat;
	a_tyAlmText : ARRAY[10000..10250] OF tyAlmTxt := [(sAlmText:='Invalid Ident While Creating Server',sRcyText:='Problem Occurred In The TCP/IP Connection. Check The Connection And Try To Reconnect.'),(sAlmText:='Setting Keep Alive Interval Time Error While Creating Server',sRcyText:='Unable To Establish Connection Between Machine. Check For Setting And Resume Operation.'),(sAlmText:='Setting Keep Alive Idle Time Error While Creating Server',sRcyText:='Unable To Establish Connection Between Machine. Check For Setting And Resume Operation.'),(sAlmText:='Setting Keep Alive Count Error While Creating Server',sRcyText:='Unable To Establish Connection Between Machine. Check For Setting And Resume Operation.'),(sAlmText:='Setting Keep Alive Error While Creating Server',sRcyText:='Unable To Establish Connection Between Machine. Check For Setting And Resume Operation.'),(sAlmText:='Setting Receive Buffer Error While Creating Server',sRcyText:='Unable To Establish Connection Between Machine. Check For Setting And Resume Operation.'),(sAlmText:='Setting Send Buffer Error While Creating Server',sRcyText:='Unable To Establish Connection Between Machine. Check For Setting And Resume Operation.'),(sAlmText:='Setting No Waiting Error While Creating Server',sRcyText:='Unable To Establish Connection Between Machine. Check For Setting And Resume Operation.'),(sAlmText:='TCP Open Port Error While Creating Server',sRcyText:='Problem Occurred In The TCP/IP Connection. Check The Connection And Try To Reconnect.'),(sAlmText:='Closing TCP Error While Creating Server',sRcyText:='Problem Occurred In The TCP/IP Connection. Check The Connection And Try To Reconnect.'),(sAlmText:='Invalid Ident While Listening Client',sRcyText:='There Was A Problem Connecting To The Server. The Server May Not Exist or It is Unavailable At This Time. Check The Connection and Try Again.'),(0),(sAlmText:='Supervisory Hermes Connection Lost',sRcyText:='There Was A Problem Connecting To The Server. The Server May Not Exist or It is Unavailable At This Time. Check The Connection and Try Again.'),(0),(sAlmText:='Invalid Ident While Receiving Data',sRcyText:='Problem Occurred In The TCP/IP Connection. Check The Connection And Try To Reconnect.'),(sAlmText:='TCP Receive Data Error While Receiving Data',sRcyText:='Problem Occurred In The TCP/IP Connection. Check The Connection And Try To Reconnect.'),(sAlmText:='Receive SetConfiguration While Supervisory In Not Connected State',sRcyText:='Receive Illegal Message.'),(sAlmText:='Receive GetConfiguration While Supervisory In Not Connected State',sRcyText:='Receive Illegal Message.'),(sAlmText:='Receive CurrConfiguration While Supervisory In Not Connected State',sRcyText:='Receive Illegal Message.'),(sAlmText:='Receive SendWorkOrderInfo While Supervisory In Not Connected State',sRcyText:='Receive Illegal Message.'),(sAlmText:='Receive QueryWorkOrderInfo While Supervisory In Not Connected State',sRcyText:='Receive Illegal Message.'),(sAlmText:='Receive BoardArrived While Supervisory In Not Connected State',sRcyText:='Receive Illegal Message.'),(sAlmText:='Receive BoardDeparted While Supervisory In Not Connected State',sRcyText:='Receive Illegal Message.'),2((0)),(sAlmText:='Receive BoardAvailable While Downstream In Service Description State',sRcyText:='Receive Illegal Message.'),(sAlmText:='Receive RevokeBoardAvailable While Downstream In Service Description State',sRcyText:='Receive Illegal Message.'),(sAlmText:='Receive ServiceDescription While Supervisory In Service Description State',sRcyText:='Receive Illegal Message.'),(sAlmText:='Receive SetConfiguration While Supervisory In Service Description State',sRcyText:='Receive Illegal Message.'),(sAlmText:='Receive GetConfiguration While Supervisory In Service Description State',sRcyText:='Receive Illegal Message.'),(sAlmText:='Receive CurrConfiguration While Supervisory In Service Description State',sRcyText:='Receive Illegal Message.'),(sAlmText:='Receive SendWorkOrderInfo While Supervisory In Service Description State',sRcyText:='Receive Illegal Message.'),(sAlmText:='Receive QueryWorkOrderInfo While Supervisory In Service Description State',sRcyText:='Receive Illegal Message.'),(sAlmText:='Receive BoardArrived While Supervisory In Service Description State',sRcyText:='Receive Illegal Message.'),(sAlmText:='Receive BoardDeparted While Supervisory In Service Description State',sRcyText:='Receive Illegal Message.'),4((0)),(sAlmText:='Receive ServiceDescription While Supervisory In Connected State',sRcyText:='Receive Illegal Message.'),(sAlmText:='Receive CurrConfiguration While Supervisory In Connected State',sRcyText:='Receive Illegal Message.'),(sAlmText:='Receive QueryWorkOrderInfo While Supervisory In Connected State',sRcyText:='Receive Illegal Message.'),(sAlmText:='Receive BoardArrived While Supervisory In Connected State',sRcyText:='Receive Illegal Message.'),(sAlmText:='Receive BoardDeparted While Supervisory In Connected State',sRcyText:='Receive Illegal Message.'),43((0)),(sAlmText:='SystemId Missing While Checking Service Description',sRcyText:='Missing Input Value For SystemId. Fill Up The Value And Resend.'),(sAlmText:='Version Missing While Checking Service Description',sRcyText:='Missing Input Value For Version. Fill Up The Value And Resend.'),(sAlmText:='SupportedFeatures Missing While Checking Service Description',sRcyText:='Missing Input Value For SupportedFeatures. Fill Up The Value And Resend.'),2((0)),(sAlmText:='NotificationCode Out Of Range While Checking Notification',sRcyText:='NotificationCode Does Not Fall Within The Expected Range.'),(sAlmText:='NotificationCode Missing While Checking Notification',sRcyText:='Missing Input Value For NotificationCode. Fill Up The Value And Resend.'),(sAlmText:='Severity Missing While Checking Notification',sRcyText:='Missing Input Value For Severity. Fill Up The Value And Resend.'),(sAlmText:='Description Missing While Checking Notification',sRcyText:='Missing Input Value For Description. Fill Up The Value And Resend.'),10((0)),(sAlmText:='Supervisory Service Description Interchange Time Out',sRcyText:='Timeout Expired Before Operation Completed. Reset And Resume Operation.'),4((0)),(sAlmText:='Get Directory Info Error While Deleting Old Log',sRcyText:='An Error Was Encountered While Getting Directory Info. Please Contact Nutek For A Possible Solution.'),(sAlmText:='Directory Read Error While Deleting Old Log',sRcyText:='An Error Was Encountered While Reading Directory. Please Contact Nutek For A Possible Solution.'),(sAlmText:='File Delete Error While Deleting Old Log',sRcyText:='An Error Was Encountered While Trying To Delete File. Please Contact Nutek For A Possible Solution.'),(sAlmText:='File Open Error While Reading Retain File',sRcyText:='An Error Was Encountered While Trying To Open File. Please Contact Nutek For A Possible Solution.'),(sAlmText:='File Read Error While Reading Retain File',sRcyText:='An Error Was Encountered While Trying To Read File. Please Contact Nutek For A Possible Solution.'),(sAlmText:='File Close Error While Reading Retain File',sRcyText:='An Error Was Encountered While Trying To Close File. Please Contact Nutek For A Possible Solution.'),(sAlmText:='File Open Error While Writting Retain File',sRcyText:='An Error Was Encountered While Trying To Open File. Please Contact Nutek For A Possible Solution.'),(sAlmText:='File Create Error While Writting Retain File',sRcyText:='An Error Was Encountered While Trying To Create File. Please Contact Nutek For A Possible Solution.'),(sAlmText:='File Write Error While Writting Retain File',sRcyText:='An Error Was Encountered While Trying To Write File. Please Contact Nutek For A Possible Solution.'),(sAlmText:='File Close Error While Writting Retain File',sRcyText:='An Error Was Encountered While Trying To Close File. Please Contact Nutek For A Possible Solution.'),(sAlmText:='Directory Does Not Exist While Writing Retain File',sRcyText:='The Directory Does Not Exist. Please Contact Nutek For A Possible Solution.'),(sAlmText:='Revoke Board Available Request To Send From Supervisory Hermes',sRcyText:='Sending Illegal Message.'),(sAlmText:='Stop Transport Request To Send From Supervisory Hermes',sRcyText:='Sending Illegal Message.'),(sAlmText:='Transport Finished Request To Send From Supervisory Hermes',sRcyText:='Sending Illegal Message.'),(sAlmText:='Board Available Request To Send From Supervisory Hermes',sRcyText:='Sending Illegal Message.'),6((0)),(sAlmText:='Check Alive Time Out',sRcyText:='Timeout Expired Before Operation Completed. Reset And Resume Operation.'),(sAlmText:='Waiting Check Alive Time Out',sRcyText:='Timeout Expired Before Operation Completed. Reset And Resume Operation.'),(sAlmText:='Check Alive Id Mismatch',sRcyText:='The Check Alive Id Value Does Not Match. Change The Value And Resend The Value.'),(sAlmText:='Machine Ready Request To Send From Supervisory Hermes',sRcyText:='Sending Illegal Message.'),(sAlmText:='Revoke Machine Ready Request To Send From Supervisory Hermes',sRcyText:='Sending Illegal Message.'),(sAlmText:='Start Transport Request To Send From Supervisory Hermes',sRcyText:='Sending Illegal Message.'),(sAlmText:='Set Configuration Request To Send From Supervisory Hermes',sRcyText:='Sending Illegal Message.'),(sAlmText:='Get Configuration Request To Send From Supervisory Hermes',sRcyText:='Sending Illegal Message.'),(sAlmText:='Current Configuration Request To Send From Supervisory Hermes',sRcyText:='Sending Illegal Message.'),(sAlmText:='Board Forecast Request To Send From Supervisory Hermes',sRcyText:='Sending Illegal Message.'),(sAlmText:='Query Board Info Request To Send From Supervisory Hermes',sRcyText:='Sending Illegal Message.'),(sAlmText:='Invalid Ident While Sending Data',sRcyText:='Invalid Ident Value.'),(sAlmText:='TCP Retry Send Data Error While Sending Data',sRcyText:='Problem Occurred In The TCP/IP Connection. Check The Connection And Try To Reconnect.'),(sAlmText:='TCP Send Data Error',sRcyText:='Problem Occurred In The TCP/IP Connection. Check The Connection And Try To Reconnect.'),(sAlmText:='Invalid Ident While Closing TCP',sRcyText:='Invalid Ident Value.'),(sAlmText:='Closing TCP Error',sRcyText:='Problem Occurred In The TCP/IP Connection. Check The Connection And Try To Reconnect.'),(sAlmText:='File Open Error While Writing Log',sRcyText:='An Error Was Encountered While Trying To Open File. Please Contact Nutek For A Possible Solution.'),(sAlmText:='File Create Error While Writing Log',sRcyText:='An Error Was Encountered While Trying To Create File. Please Contact Nutek For A Possible Solution.'),(sAlmText:='Get File Info Error While Writing Log',sRcyText:='An Error Was Encountered While Getting File Info. Please Contact Nutek For A Possible Solution.'),(sAlmText:='File Write Error While Writing Log',sRcyText:='An Error Was Encountered While Trying To Write File. Please Contact Nutek For A Possible Solution.'),(sAlmText:='File Close Error While Writing Log',sRcyText:='An Error Was Encountered While Trying To Close File. Please Contact Nutek For A Possible Solution.'),(sAlmText:='Directory Does Not Exist While Writing Log',sRcyText:='The Directory Does Not Exist.Please Contact Nutek For A Possible Solution.'),(sAlmText:='Invalid Ident While Closing TCP',sRcyText:='Invalid Ident Value.'),(sAlmText:='Closing TCP Error',sRcyText:='Problem Occurred In The TCP/IP Connection. Check The Connection And Try To Reconnect.'),3((0)),(sAlmText:='Send Board Info Request To Send From Supervisory Hermes',sRcyText:='Sending Illegal Message.'),(sAlmText:='Query Work Order Info Request To Send From Supervisory Hermes',sRcyText:='Sending Illegal Message.'),(sAlmText:='Send Work Order Info Request To Send From Supervisory Hermes',sRcyText:='Sending Illegal Message.'),(sAlmText:='Board Arrived Request To Send From Supervisory Hermes',sRcyText:='Sending Illegal Message.'),(sAlmText:='Board Depated Request To Send From Supervisory Hermes',sRcyText:='Sending Illegal Message.'),(sAlmText:='QueryId Mismatch While Checking SendWorkOrderInfo and QueryWorkOrderInfo',sRcyText:='The QueryId Value Does Not Match. Change The Value And Resend The Value.'),(sAlmText:='QueryId Missing While Checking Send Work Order Info',sRcyText:='Missing Input Value For QueryId. Fill Up The Value And Resend.'),20((0)),(sAlmText:='File Open Error While Writing Config File',sRcyText:='An Error Was Encountered While Trying To Open File. Please Contact Nutek For A Possible Solution.'),(sAlmText:='File Create Error While Writing Config File',sRcyText:='An Error Was Encountered While Trying To Create File. Please Contact Nutek For A Possible Solution.'),(sAlmText:='File Write Error While Writing Config File',sRcyText:='An Error Was Encountered While Trying To Write File. Please Contact Nutek For A Possible Solution.'),(sAlmText:='File Close Error While Writing Config File',sRcyText:='An Error Was Encountered While Trying To Close File. Please Contact Nutek For A Possible Solution.'),(sAlmText:='Directory Does Not Exist While Writing Config File',sRcyText:='The Directory Does Not Exist. Please Contact Nutek For A Possible Solution.'),9((0)),(sAlmText:='File Open Error While Reading Loader Work Order Retain File',sRcyText:='An Error Was Encountered While Trying To Open File. Please Contact Nutek For A Possible Solution.'),(sAlmText:='File Read Error While Reading Loader Work Order Retain File',sRcyText:='An Error Was Encountered While Trying To Read File. Please Contact Nutek For A Possible Solution.'),(sAlmText:='File Close Error While Reading Loader Work Order Retain File',sRcyText:='An Error Was Encountered While Trying To Close File. Please Contact Nutek For A Possible Solution.'),(sAlmText:='File Open Error While WrittingLoader Work Order  Retain File',sRcyText:='An Error Was Encountered While Trying To Open File. Please Contact Nutek For A Possible Solution.'),(sAlmText:='File Create Error While Writting Loader Work Order Retain File',sRcyText:='An Error Was Encountered While Trying To Create File. Please Contact Nutek For A Possible Solution.'),(sAlmText:='File Write Error While Writting Loader Work Order Retain File',sRcyText:='An Error Was Encountered While Trying To Write File. Please Contact Nutek For A Possible Solution.'),(sAlmText:='File Close Error While Writting Loader Work Order  Retain File',sRcyText:='An Error Was Encountered While Trying To Close File. Please Contact Nutek For A Possible Solution.'),(sAlmText:='Directory Does Not Exist While Loader Work Order Writing Retain File',sRcyText:='The Directory Does Not Exist. Please Contact Nutek For A Possible Solution.'),(sAlmText:='File Open Error While Reading Loader Loaded Work Order Retain File',sRcyText:='An Error Was Encountered While Trying To Open File. Please Contact Nutek For A Possible Solution.'),(sAlmText:='File Read Error While Reading Loader Loaded Work Order Retain File',sRcyText:='An Error Was Encountered While Trying To Read File. Please Contact Nutek For A Possible Solution.'),(sAlmText:='File Close Error While Reading Loader Loaded Work Order Retain File',sRcyText:='An Error Was Encountered While Trying To Close File. Please Contact Nutek For A Possible Solution.'),(sAlmText:='File Open Error While Writting Loader Loaded Work Order Retain File',sRcyText:='An Error Was Encountered While Trying To Open File. Please Contact Nutek For A Possible Solution.'),(sAlmText:='File Create Error While Writting Loaded Work Order Retain File',sRcyText:='An Error Was Encountered While Trying To Create File. Please Contact Nutek For A Possible Solution.'),(sAlmText:='File Write Error While Writting Loader Loaded Work Order Retain File',sRcyText:='An Error Was Encountered While Trying To Write File. Please Contact Nutek For A Possible Solution.'),(sAlmText:='File Close Error While Writting Loader Loaded Work Order Retain File',sRcyText:='An Error Was Encountered While Trying To Close File. Please Contact Nutek For A Possible Solution.'),(sAlmText:='Directory Does Not Exist While Writing Loader Loaded Work Order Retain File',sRcyText:='The Directory Does Not Exist. Please Contact Nutek For A Possible Solution.'),(sAlmText:='File Open Error While Reading Bypass Work Order Retain File',sRcyText:='An Error Was Encountered While Trying To Open File. Please Contact Nutek For A Possible Solution.'),(sAlmText:='File Read Error While Reading Bypass  Work Order Retain File',sRcyText:='An Error Was Encountered While Trying To Read File. Please Contact Nutek For A Possible Solution.'),(sAlmText:='File Close Error While Reading Bypass Work Order Retain File',sRcyText:='An Error Was Encountered While Trying To Close File. Please Contact Nutek For A Possible Solution.'),(sAlmText:='File Open Error While Writting Bypass Work Order Retain File',sRcyText:='An Error Was Encountered While Trying To Open File. Please Contact Nutek For A Possible Solution.'),(sAlmText:='File Create Error While Writting Bypass  Work Order Retain File',sRcyText:='An Error Was Encountered While Trying To Create File. Please Contact Nutek For A Possible Solution.'),(sAlmText:='File Write Error While Writting Bypass  Work Order Retain File',sRcyText:='An Error Was Encountered While Trying To Write File. Please Contact Nutek For A Possible Solution.'),(sAlmText:='File Close Error While Writting Bypass  Work Order Retain File',sRcyText:='An Error Was Encountered While Trying To Close File. Please Contact Nutek For A Possible Solution.'),(sAlmText:='Directory Does Not Exist While Writing Bypass  Work Order Retain File',sRcyText:='The Directory Does Not Exist. Please Contact Nutek For A Possible Solution.'),0,26((0))];
END_VAR
(**)
(*Local Output*)
VAR
	bConnected : BOOL;
	bTest : BOOL;
	bTest1 : BOOL;
	bTest2 : BOOL;
	bHandshakeDone : BOOL;
	sInternalSnd : STRING[65535];
	bFileNotFound : BOOL := FALSE;
	bWriteConfig : BOOL := FALSE;
	bUpdateUIData : BOOL := FALSE;
END_VAR
(**)
(*Local Input*)
VAR
	udiRstErr : UDINT := 0;
	bPrep : BOOL := TRUE;
	bEn : BOOL := TRUE;
	bDis : BOOL := FALSE;
	tyParam : tyHermesSvyParam;
	sIPAddr : STRING[15] := '192.168.0.100';
	a_usiMacAddr : ARRAY[0..5] OF USINT := [6(0)];
	tyDTStructure : DTStructure := (year:=2020,month:=11,day:=05,wday:=05,hour:=21,minute:=28,second:=30,millisec:=123,microsec:=456);
	dtCurrDT : DATE_AND_TIME := DT#2019-02-23-12:30:50;
	sMcId : STRING[80] := '';
	sMagazineId : STRING[80] := '';
	iSlotId : INT;
	sBarcode : STRING[254] := '';
	eBoardTransfer1 : eHermesBoardTransfer := HermesTransferred;
	eBoardTransfer2 : eHermesBoardTransfer := HermesTransferred;
	eBoardTransfer3 : eHermesBoardTransfer := HermesTransferred;
	eBoardTransfer4 : eHermesBoardTransfer := HermesTransferred;
	sVersion : STRING[7] := '1.3';
	sWorkOrderId : STRING[80] := '';
	sBatchId : STRING[80] := '';
	sRecipeNm : STRING[254] := '';
	udiSndBffrSize : UDINT := 65536;
	udiRcvBffrSize : UDINT := 65536;
	udiAliveIdleTimeInSec : UDINT := 5;
	tConnTimeOut : TIME := T#30s;
	diTransferInTO : DINT := 30000;
	bNewBrdAvl : BOOL := FALSE;
	bOpsRun : BOOL := FALSE;
	udiFileKeepDay : UDINT := 30;
	sConfigFileName : STRING[80] := 'SvyHermes.dat';
	sProgNm : STRING[15] := 'SvyHermes';
	sRetainFileName : STRING[80] := 'WorkOrder.dat';
	sRetainFileName1 : STRING[80] := 'LoaderSendWorkOrder.dat';
	sRetainFileName2 : STRING[80] := 'LoaderLoadedSendWorkOrder.dat';
	sRetainFileName3 : STRING[80] := 'BypassSendWorkOrder.dat';
	bNtSettingsLoadDone : BOOL := TRUE;
	bSvyPrep : BOOL := FALSE;
	bSvyEn : BOOL := FALSE;
	sInfoMsg : STRING[200];
	sInfoMsg1 : STRING[200];
	sInfoMsg2 : STRING[200];
	sInfoMsg3 : STRING[200];
	sInfoMsg4 : STRING[200];
	bEndSen : BOOL := FALSE;
	tyHermesCurrConfiguration : tyHermesConfiguration;
	bQueryWorkOrderInfo : BOOL := TRUE;
	bAcceptCondition : BOOL;
	bAllZonesEmpty : BOOL;
	bDeleteWorkOrder : BOOL;
	bFirstMcIntheLine : BOOL;
	bUSHermesStopTransportSnd1 : BOOL;
	bUSHermesStopTransportSnd2 : BOOL;
	bUSHermesStopTransportSnd3 : BOOL;
	bUSHermesStopTransportSnd4 : BOOL;
	bDSHermesTransportFinishedSnd1 : BOOL;
	bDSHermesTransportFinishedSnd2 : BOOL;
	bDSHermesTransportFinishedSnd3 : BOOL;
	bDSHermesTransportFinishedSnd4 : BOOL;
	tyUSHermesBoardArrivedData1 : tyHermesBoardAvailable;
	tyUSHermesBoardArrivedData2 : tyHermesBoardAvailable;
	tyUSHermesBoardArrivedData3 : tyHermesBoardAvailable;
	tyUSHermesBoardArrivedData4 : tyHermesBoardAvailable;
	tyDSHermesBoardDepartedData1 : tyHermesBoardAvailable;
	tyDSHermesBoardDepartedData2 : tyHermesBoardAvailable;
	tyDSHermesBoardDepartedData3 : tyHermesBoardAvailable;
	tyDSHermesBoardDepartedData4 : tyHermesBoardAvailable;
	bInternalUse : BOOL;
	sInternalRcv : STRING[65535];
END_VAR
(**)
(*Local*)
VAR
	bRstErr : BOOL;
	udiRstErrOld : UDINT;
	bInitDone : BOOL;
	bInitialDone : BOOL;
	bRun : BOOL;
	bStop : BOOL;
	bRstConnection : BOOL;
	bRstState : BOOL;
	bSndWorkOrderInfo : BOOL;
	bRcvWorkOrderInfo1 : BOOL;
	bRcvWorkOrderInfo2 : BOOL;
	bRcvWorkOrderInfo3 : BOOL;
	bRcvBypassWorkOrderInfo2 : BOOL;
	bRstWorkOrderInfo : BOOL;
	bFoundIndexUS1 : BOOL;
	bFoundIndexUS2 : BOOL;
	bFoundIndexUS3 : BOOL;
	bFoundIndexUS4 : BOOL;
	bFoundIndexDS1 : BOOL;
	bFoundIndexDS2 : BOOL;
	bFoundIndexDS3 : BOOL;
	bFoundIndexDS4 : BOOL;
	udiFoundIndexUS1 : UDINT;
	udiFoundIndexUS2 : UDINT;
	udiFoundIndexUS3 : UDINT;
	udiFoundIndexUS4 : UDINT;
	udiFoundIndexDS1 : UDINT;
	udiFoundIndexDS2 : UDINT;
	udiFoundIndexDS3 : UDINT;
	udiFoundIndexDS4 : UDINT;
	k : UDINT := 0;
	kk : UDINT := 0;
	j : INT := 1;
	jj : INT := 2;
	jjj : INT := 3;
	jjjj : INT := 4;
	udiSvrIdent : UDINT;
	udiClntIdent : UDINT;
	udiClntIdentExtra : UDINT;
	udiXMLTableWriteIdx : UDINT;
	udiMsgSendBffr : UDINT;
	udiSndMsgLen : UDINT;
	sSnd : STRING[65535];
	sRcv : STRING[65535];
	a_tyXMLTableDataRcv : ARRAY[0..200] OF tyXMLTableDat;
	a_tyXMLTableDataSnd : ARRAY[0..200] OF tyXMLTableDat;
	a_eMsgSend : ARRAY[0..50] OF eHermesMsgType;
	tyMsgTypeRcv : tyHermesMsgType;
	tyCheckAliveSnd : tyHermesCheckAlive;
	tyCheckAlivePingSnd : tyHermesCheckAlive;
	tyCheckAlivePongSnd : tyHermesCheckAlive;
	tyCheckAliveRcv : tyHermesCheckAlive;
	tyCheckAlivePingRcv : tyHermesCheckAlive;
	tyCheckAlivePongRcv : tyHermesCheckAlive;
	tyServiceDescriptionRcv : tyHermesServiceDescription;
	tySServiceDescriptionSnd : tyHermesSServiceDescription;
	tySServiceDescriptionRcv : tyHermesSServiceDescription;
	tyNotificationSnd : tyHermesNotification;
	tyNotificationRcv : tyHermesNotification;
	tyBoardAvailableRcv : tyHermesBoardAvailable;
	tyMachineReady : tyHermesMachineReady;
	tyStartTransport : tyHermesStartTransport;
	tyStopTransport : tyHermesStopTransport;
	tyTransportFinished : tyHermesTransportFinished;
	tySetConfiguration : tyHermesSetConfiguration;
	tySetConfigurationRcv : tyHermesSetConfiguration;
	tySetConfigurationModified : tyHermesSetConfiguration;
	tyCurrentConfigurationRcv : tyHermesCurrentConfiguration;
	tyCurrentConfigurationSnd : tyHermesCurrentConfiguration;
	tyBoardForecast : tyHermesBoardForecast;
	tyBoardArrivedRcv : tyHermesBoardArrived;
	tyBoardArrived1 : tyHermesBoardArrived;
	tyBoardArrived2 : tyHermesBoardArrived;
	tyBoardArrived3 : tyHermesBoardArrived;
	tyBoardArrived4 : tyHermesBoardArrived;
	tyBoardDepartedRcv : tyHermesBoardDeparted;
	tyBoardDeparted1 : tyHermesBoardDeparted;
	tyBoardDeparted2 : tyHermesBoardDeparted;
	tyBoardDeparted3 : tyHermesBoardDeparted;
	tyBoardDeparted4 : tyHermesBoardDeparted;
	tyQueryBoardInfo : tyHermesQueryBoardInfo;
	tySendBoardInfo : tyHermesSendBoardInfo;
	tyQueryWorkOrderInfo : tyHermesQueryWorkOrderInfo; (*Query For Loader Mode*)
	tyQueryBypassWorkOrderInfo : tyHermesQueryWorkOrderInfo; (*Query For Bypass mode*)
	tyReplyWorkOrderInfo : tyHermesReplyWorkOrderInfo;
	tySendWorkOrderInfoAcc : tyHermesSendWorkOrderInfo;
	tySendBypassWorkOrderInfoAcc : tyHermesSendWorkOrderInfo;
	tySendWorkOrderInfoRcv : tyHermesSendWorkOrderInfo;
	tyDummySendWorkOrderInfoRcv : tyHermesSendWorkOrderInfo;
	tySendWorkOrderInfoNewAcc : tyHermesSendWorkOrderInfo;
	fbCreateSvr : fbTCPCreateSvr;
	fbListen : fbTCPListen;
	fbRcv : fbTCPRcv;
	fbSend : fbTCPSnd;
	fbCloseSvr : fbTCPClose;
	fbCloseClnt : fbTCPClose;
	fbParseXMLTable : fbHermesParseXMLTable;
	fbCheckAlive : fbHermesCheckAlive;
	fbCheckAliveSendPing : fbHermesCheckAliveSendPing;
	fbCheckAliveRcvPing : fbHermesCheckAliveRcvPing;
	fbSequenceSvy : fbHermesSequenceSvy;
	fbSequenceTO : fbHermesSequenceSvyTO;
	eStatOld : eHermesAction := HermesActIdle;
	tyParamOld : tyHermesSvyParam;
	udiLogCntr : UDINT := 1;
	udiWriteLogCntr : UDINT := 1;
	a_sLogList : ARRAY[1..10] OF STRING[65535];
	sDT : STRING[80];
	dtCurrDTTemp : DATE_AND_TIME;
	fbFileAppend1 : fbFileFullAppend;
	fbFileOldDel1 : fbFileOldDel;
	fbFileRead1 : fbFileFullRead;
	fbFileWrite1 : fbFileFullWrite;
	fbFileRead2 : fbFileFullRead;
	fbFileWrite2 : fbFileFullWrite;
	fbFileRead3 : fbFileFullRead;
	fbFileWrite3 : fbFileFullWrite;
	fbFileRead4 : fbFileFullRead;
	fbFileWrite4 : fbFileFullWrite;
	fbDelayTm : TON;
	fbDelayTm1 : TON;
	udiTargetAddress : UDINT := 0;
	udiTargetAddress1 : UDINT := 0;
	udiSizeAddress : UDINT := 0;
	udiSizeAddress1 : UDINT := 0;
	udiRetainDataAddr : UDINT;
	udiRetainDataLen : UDINT;
	udiLoaderRetainDataAddr0 : UDINT;
	udiLoaderRetainDataLen0 : UDINT;
	udiLoaderRetainDataAddr1 : UDINT;
	udiLoaderRetainDataLen1 : UDINT;
	udiBypassRetainDataAddr0 : UDINT;
	udiBypassRetainDataLen0 : UDINT;
	diReqWidthInUM : DINT;
	diReqLoaderWidthInUM : DINT;
	iWriteLogStep : INT := 0;
	udiModuleNum : UDINT := 6761;
	a_bQueryQueue : ARRAY[0..3] OF BOOL;
	i2 : USINT;
	sMagPos : STRING[80] := '';
	uiMilliSecOld : UINT;
END_VAR
(*Local priority param*)
VAR
	bGUIDInserted : ARRAY[1..3] OF BOOL;
	a_MagGUID : ARRAY[1..3] OF STRING[80];
END_VAR
VAR RETAIN
	a_MagAccOrder : ARRAY[1..3] OF USINT; (*priority (output)*)
END_VAR
VAR
	usiMagPrior : ARRAY[1..3] OF USINT := [1,2,3];
	usiMagRun : ARRAY[1..3] OF USINT;
	usiSum : ARRAY[1..3] OF USINT;
	usiMagOrderPos : USINT;
	i : USINT;
	i1 : USINT;
END_VAR
```

#### Act_Background_CmpParamRcv.st
```iecst
(** 2021-08-01 **)
ACTION Act_Background_CmpParamRcv:

	IF eStatus2 <> Error THEN

		IF tySServiceDescriptionRcv.tyAvl.tySupportedFeatures.bFeatureSendWorkOrderInfo = TRUE AND p_tyParam.bFeatureQueryWorkOrderInfo THEN
				                                                                          //ADD
			IF tyMsgTypeRcv.bSendWorkOrderInfo = TRUE AND (p_bQueryWorkOrderInfo OR tyQueryWorkOrderInfo.tyAvl.bQueryId) THEN
//				udiStatus2	:= fHermesChkParamSWQW(tySendWorkOrderInfoRcv , tyQueryWorkOrderInfo);
//				udiStatus5  := fHermesChkParamSWBQW(tySendWorkOrderInfoRcv , tyQueryBypassWorkOrderInfo);	          //ADD

				IF udiStatus2 <> 0 AND udiStatus5 <> 0 THEN
					eStatus2	:= Error;

					IF udiStatus2 = 2767 THEN
						udiStatus2	:= 10164;	//QueryId Mismatch While Checking SendWorkOrderId & QueryWorkOrderId
					ELSIF udiStatus5 = 2767  THEN
						udiStatus2	:= 10164;	//QueryId Mismatch While Checking SendWorkOrderId & QueryWorkOrderId
					ELSIF udiStatus2 = 2768 THEN
						udiStatus2	:= 10165;	//QueryId Missing While Checking SendWorkOrderId & QueryWorkOrderId
					ELSIF udiStatus5 = 2768 THEN
						udiStatus2	:= 10165;	//QueryId Missing While Checking SendWorkOrderId & QueryWorkOrderId
					END_IF

					fHermesAddOneMsgSend(ADR(a_eMsgSend) , ADR(udiMsgSendBffr) , HermesMsgTypeNotification);

					tyNotificationSnd.tyAvl.bSeverity			:= TRUE;
					tyNotificationSnd.tyAvl.bNotificationCode	:= TRUE;
					tyNotificationSnd.tyAvl.bDescription		:= TRUE;
					tyNotificationSnd.tyData.eSeverity			:= HermesSeverityError;
					tyNotificationSnd.tyData.iNotificationCode	:= UDINT_TO_INT(udiStatus2);
					tyNotificationSnd.tyData.sDescription		:= a_tyAlmText[udiStatus2].sAlmText;

					tyMsgTypeRcv.bSendWorkOrderInfo := FALSE; //reset, else latching
				END_IF
			END_IF
		END_IF
	END_IF

		END_ACTION
```

#### Act_Background_ProcessData.st
```iecst
(** 2021-08-01 **)
ACTION Act_Background_ProcessData:

	//Write Config into "Hermes"
	fbDelayTm(IN := bWriteConfig, PT := T#0.5S); //Small Delay 0.5s to let Hermes take the Data, before WriteConfig

	IF fbDelayTm.Q THEN

		eHermesAct := HermesActWriteConfig;
		eMcParamAct := McParamActWrite;

		IF p_eHermesStatus = Done AND p_eHermesStat = HermesActWriteConfig AND p_eMcParamStat = McParamActWrite AND p_eMcParamStatus = Done THEN

		eMcParamAct     := McParamActIdle;
	   	eHermesAct		:= HermesActIdle;
		bWriteConfig    := FALSE;
		bUpdateUIData   := TRUE;
		fbDelayTm(IN := FALSE);
		tyInfoData.sProgNm		:= p_sProgNm;
		tyInfoData.udiCode		:= 10000;
		tyInfoData.eSeverity	:= AlmSeverityInfo;
		tyInfoData.sAlmMsg		:= p_sInfoMsg;

	    ELSIF  (p_eHermesStatus = Error AND p_eHermesStat = HermesActWriteConfig) OR (p_eMcParamStat = McParamActWrite AND p_eMcParamStatus = Error)  THEN

			eMcParamAct     := McParamActIdle;
		    eHermesAct		:= HermesActIdle;
		    bWriteConfig    := FALSE;
		    bUpdateUIData   := FALSE;
			fbDelayTm(IN := FALSE);

			fHermesAddOneMsgSend(ADR(a_eMsgSend) , ADR(udiMsgSendBffr) , HermesMsgTypeNotification);

			udiStatus2 := 10199; //SetConfiguration Failed, Please Send Again
			tyNotificationSnd.tyAvl.bSeverity			:= TRUE;
			tyNotificationSnd.tyAvl.bNotificationCode	:= TRUE;
			tyNotificationSnd.tyAvl.bDescription		:= TRUE;
			tyNotificationSnd.tyData.eSeverity			:= HermesSeverityFatalError;
			tyNotificationSnd.tyData.iNotificationCode	:= UDINT_TO_INT(udiStatus2);
			tyNotificationSnd.tyData.sDescription		:= a_tyAlmText[udiStatus2].sAlmText;

		END_IF
	END_IF

	//Update UI
	IF bUpdateUIData THEN
		tyInfoData.sProgNm		:= p_sProgNm;
		tyInfoData.udiCode		:= 10000;
		tyInfoData.eSeverity	:= AlmSeverityInfo;
		tyInfoData.sAlmMsg		:= p_sInfoMsg;
	END_IF

	//Auto Reset
	fbDelayTm1(IN := bUpdateUIData , PT := T#2S); //Auto reset the Info Msg C0009 page. No need press.
	IF fbDelayTm1.Q = TRUE THEN

		//Clear Info Message
		tyInfoData.sProgNm		:= '';
		tyInfoData.udiCode		:= 0;
		tyInfoData.eSeverity	:= AlmSeverityNA;
		tyInfoData.sAlmMsg		:= '';

		bUpdateUIData  := FALSE;
		bFoundIndexUS1 := FALSE;
		bFoundIndexUS2 := FALSE;
		bFoundIndexUS3 := FALSE;
		bFoundIndexUS4 := FALSE;
		bFoundIndexDS1 := FALSE;
		bFoundIndexDS2 := FALSE;
		bFoundIndexDS3 := FALSE;
		bFoundIndexDS4 := FALSE;

		fbDelayTm1(IN := FALSE);
	END_IF

	//BatchId from Supervisory System
	sBatchId := tySendWorkOrderInfoAcc.tyData.sBatchId;

	//Retain sWorkOrderId for machine power cycle
	p_udiRetainDataAddr	:= ADR(sWorkOrderId);
	p_udiRetainDataLen	:= SIZEOF(sWorkOrderId);

	//Write Retain
//	IF EDGEPOS(bRcvWorkOrderInfo1) THEN
//    	sWorkOrderId := tySendWorkOrderInfoAcc.tyData.sWorkOrderId; //Receive from Svy
//		p_eAct := HermesActWriteRetain;

	IF EDGEPOS(bRetainNewAcc) THEN
    	sWorkOrderId := tySendWorkOrderInfoNewAcc.tyData.sWorkOrderId; //Receive from Svy
		p_eAct := HermesActWriteRetain;

	ELSIF EDGENEG(p_bSvyEn = TRUE) OR EDGENEG(p_bSvyPrep = TRUE) THEN
		sWorkOrderId := ''; //Empty if Supervisory Hermes disable
		p_eAct := HermesActWriteRetain;

	ELSIF EDGENEG(p_tyHermesConfiguration.tySvyParam.bFeatureQueryWorkOrderInfo = TRUE) THEN
		sWorkOrderId := ''; //Empty if no support
		p_eAct := HermesActWriteRetain;

	ELSIF EDGEPOS(p_bDeleteWorkOrder) THEN
		sWorkOrderId := ''; //Delete from UI
	//	tySendWorkOrderInfoNewAcc := tyDummySendWorkOrderInfoRcv;
		tySendWorkOrderInfoAcc := tyDummySendWorkOrderInfoRcv;
		p_eAct := HermesActWriteRetain;
		p_bUIDeleteWorkOrder := FALSE; //bi-dir
		p_bAutoRcpCurrDeleteSendWO := FALSE; //bi-dir
		p_bDeleteWorkOrder := FALSE;
	END_IF

	//Retain tySendWorkOrderInfoAcc (Loader Accept data)
	p_udiLoaderRetainDataAddr0	:= ADR(tySendWorkOrderInfoAcc);
	p_udiLoaderRetainDataLen0   := SIZEOF(tySendWorkOrderInfoAcc);

	//Retain tySendWorkOrderInfoNewAcc (Loader loaded Accept data)
	p_udiLoaderRetainDataAddr1	:= ADR(tySendWorkOrderInfoNewAcc);
	p_udiLoaderRetainDataLen1   := SIZEOF(tySendWorkOrderInfoNewAcc);

     //Retain tySendBypassWorkOrderInfoAcc (Bypass Accept data)
	p_udiBypassRetainDataAddr0	:= ADR(tySendBypassWorkOrderInfoAcc);
	p_udiBypassRetainDataLen0   := SIZEOF(tySendBypassWorkOrderInfoAcc);

	IF EDGEPOS (bRcvWorkOrderInfo1) THEN
		p_eAct := HermesActWriteRetainSendWO1;

	ELSIF EDGEPOS (bRetainNewAcc OR p_bDeleteWorkOrder) THEN
		p_eAct := HermesActWriteRetainSendWO2;

	ELSIF EDGEPOS (bRcvWorkBypassOrderInfo) THEN
		p_eAct := HermesActWriteRetainSendWO3;
	END_IF

	IF eStatus = Done AND eStat = HermesActWriteRetain THEN
		p_eAct		:= HermesActIdle;
	ELSIF eStatus = Done AND eStat = HermesActWriteRetainSendWO1 THEN
		p_eAct		:= HermesActIdle;
	ELSIF eStatus = Done AND eStat = HermesActWriteRetainSendWO2 THEN
		p_eAct		:= HermesActIdle;
	ELSIF eStatus = Done AND eStat = HermesActWriteRetainSendWO3 THEN
		p_eAct		:= HermesActIdle;
	END_IF

//	//Testing -> Read Retain
//	IF EDGEPOS(bTest) THEN
//		p_eAct := HermesActReadRetain;
//	END_IF
//
//	IF eStatus = Done AND eStat = HermesActReadRetain THEN
//		p_eAct		:= HermesActIdle;
//	END_IF

END_ACTION
```
